% RSLogix 500 project LANLOGIX_BR.RSS, saved by version 12.00.00.00 %
PROJECT "LANLOGIX"    % processor: MicroLogix 1400; MAIN_PROG %

PROGRAM FILES
  LAD 2 "MAIN"  69 rungs
  LAD 4 "MODE SEL"  18 rungs
  LAD 5 "FILM"  6 rungs
  LAD 6 "PROFILES"  56 rungs
  LAD 7 "OPTIONS"  34 rungs
  LAD 8 "CONSTANTS"  5 rungs
  LAD 9 "WRAP CYCLE"  36 rungs
  LAD 10 "OUTPUTS"  46 rungs
  LAD 11 "INPUTS"  77 rungs
  LAD 12 "ROTATION"  44 rungs
  LAD 13 "CARRIAGE"  45 rungs
  LAD 14 "MPS"  23 rungs
  LAD 15 "CUTTER ASM"  18 rungs
  LAD 16 "FILM CLAMP"  15 rungs
  LAD 17 "HOT WIRE"  9 rungs
  LAD 19 "TSD"  37 rungs  % Top Sheet Dispenser %
  LAD 27 "CONV IN 3"  22 rungs
  LAD 28 "CONV IN 2"  22 rungs
  LAD 29 "CONV IN 1"  23 rungs
  LAD 30 "CONV WRAPZ"  29 rungs
  LAD 31 "CONV EX 1"  23 rungs
  LAD 32 "CONV EX 2"  22 rungs
  LAD 33 "CONV EX 3"  22 rungs
  LAD 41 "CONV INTLK"  4 rungs
  LAD 42 "GATE IN"  15 rungs  % Infeed Gate %
  LAD 43 "GATE EX"  15 rungs  % Exit Gate %
  LAD 45 "LOAD LIFT"  12 rungs
  LAD 49 "SECURITY"  11 rungs
  LAD 50 "HMI"  30 rungs
  LAD 52 "CYCLE INFO"  20 rungs
  LAD 98 "WARNINGS"  19 rungs
  LAD 99 "MESSAGES"  28 rungs
  LAD 100 "ALARMS"  36 rungs
  LAD 101 "MAINT"  20 rungs
  LAD 115 "PDATA"  22 rungs  % Production Data %
  LAD 116 "PCHART"  26 rungs  % Production Chart %
  LAD 117 "CDATA"  6 rungs  % Load Containment Data %
  LAD 214 "MPS CALC"  8 rungs
  LAD 250 "VFD MODBUS"  34 rungs
  LAD 251 "MODBUS"  7 rungs
  LAD 255 "HSC PFN"  2 rungs

DATA FILES
  O0 OUTPUT  8 elements
  I1 INPUT  11 elements
  S2 STATUS  66 elements
  B3 BINARY  110 elements
  T4 TIMER  251 elements
  C5 COUNTER  1 elements
  R6 CONTROL  1 elements
  N7 INTEGER  210 elements
  F8 FLOAT  40 elements
  F9 C FORCE  50 elements
  N10 OUTPUT MAP  120 elements
  N11 INPUT MAP  120 elements
  B12 BINARY  120 elements
  B13 BINARY  120 elements
  N14 LG  250 elements
  N15 OPTIONS  15 elements
  N16 SECURITY  10 elements
  N17 MESSAGING  50 elements
  N19 TRACKING  210 elements
  N20 FILM  30 elements
  N21 PROFILES  50 elements
  F22 PROF CALCS  15 elements
  L25 LONG  11 elements
  F26 ICF MAP  16 elements
  N28 TEMP PROF  50 elements  % Temporary Profile %
  N29 INPUT PROF  50 elements  % HMI Input Profile %
  N30 DEFAULT  50 elements  % Default Profile %
  N31 PROFILE 1  50 elements  % Profile 1 %
  N32 PROFILE 2  50 elements  % Profile 2 %
  N33 PROFILE 3  50 elements  % Profile 3 %
  N34 PROFILE 4  50 elements  % Profile 4 %
  N35 PROFILE 5  50 elements  % Profile 5 %
  N36 PROFILE 6  50 elements  % Profile 6 %
  N37 PROFILE 7  50 elements  % Profile 7 %
  N38 PROFILE 8  50 elements  % Profile 8 %
  N39 PROFILE 9  50 elements  % Profile 9 %
  N40 CURRENT  50 elements
  N41 PROFILECAL  28 elements
  ST43 PROFILESTR  10 elements
  ST46 PROFILES  15 elements
  B48 PROF WARN  8 elements
  N49 PROFWARNCH  10 elements
  N50 HMI OUTPUT  256 elements
  N51 HMI INPUT  125 elements
  B60 FAULT  255 elements  % Fault Overflow Trap %
  N80 E_NET_IN  1 elements
  N81 E_NET_OUT  1 elements
  N92 WARNCOPY  10 elements
  N93 WARN BUF  10 elements  % WARNING BUFFER %
  N94 WARN LIST  10 elements  % WARNINGS LIST %
  N95 WARNINGS  10 elements  % WARNINGS %
  N96 ALARMCOPY  50 elements
  N97 ALARM BUF  14 elements  % ALARMS BUFFER %
  N98 ALARM ACT  10 elements  % ALARM ACTIVE %
  N99 ALARM LIST  14 elements  % ALARM LIST %
  N100 ALARMS  50 elements
  N101 MAINT  30 elements
  L102 MAINT1  5 elements
  N103 MAINT2  20 elements
  N110 CDATA  40 elements  % Load Containment Data %
  N111 CDATA1  240 elements  % Load Containment Data Array 1 %
  F112 CDATA2  120 elements  % Load Containment Data Array 2 %
  N115 PDATA  20 elements  % Production Data Control %
  N116 PDATA1  160 elements  % Production Data Array 1 %
  N117 PDATA2  160 elements  % Production Data Array 2 %
  N118 PDATA3  160 elements  % Production Data Array 3 %
  N119 PDATALPH  60 elements  % Production Data Loads/Breaks Per Hour %
  N120 PDATALPR  30 elements  % Production Data Loads Per Film Roll %
  L121 PDATARPR  40 elements  % Production Data Revolutions Per Film Rolls %
  N122 PDATACHART  100 elements  % Production Data Chart %
  N170   3 elements
  N200 MODBUS  50 elements
  MG201 MODBUS MSG  5 elements
  N210 MODBUS OUT  250 elements
  N211 MODBUS IN  250 elements
  ST255 VERSION  1 elements

LADDER 2 "MAIN"
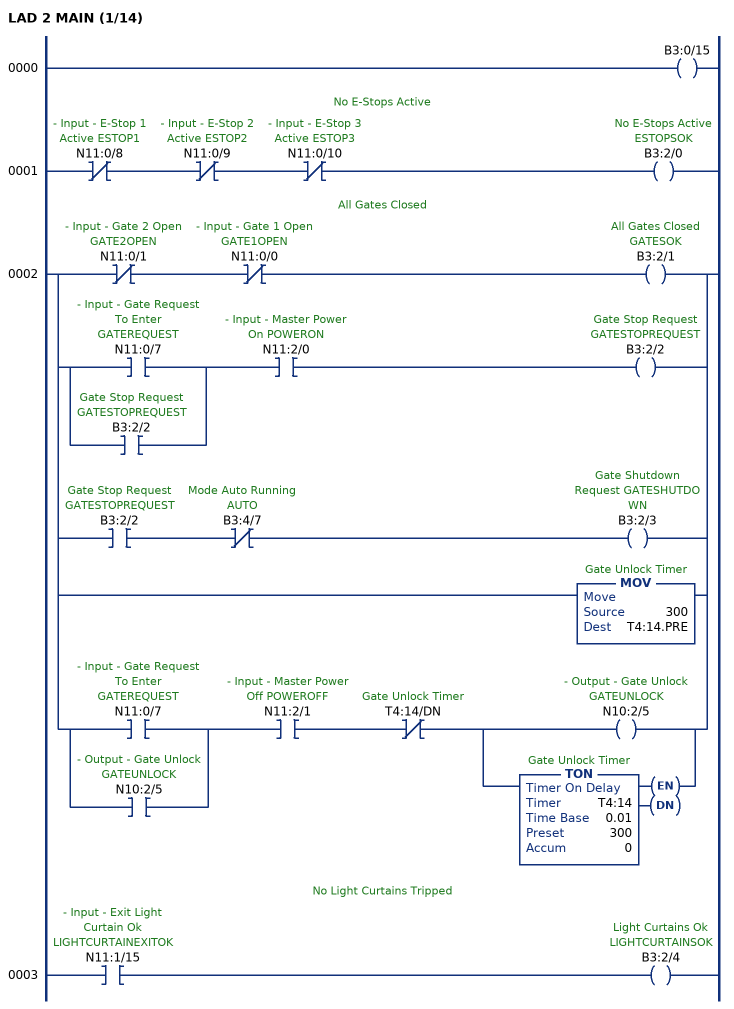
% Rung: 0 %
SOR OTE B3:0/15 EOR
% Rung: 1 %
% No E-Stops Active %
SOR XIO N11:0/8 XIO N11:0/9 XIO N11:0/10 OTE B3:2/0 EOR
%   N11:0/8  ESTOP1  "- Input - E-Stop 1 Active" %
%   N11:0/9  ESTOP2  "- Input - E-Stop 2 Active" %
%   N11:0/10  ESTOP3  "- Input - E-Stop 3 Active" %
%   B3:2/0  ESTOPSOK  "No E-Stops Active" %
% Rung: 2 %
% All Gates Closed %
SOR BST XIO N11:0/1 XIO N11:0/0 OTE B3:2/1 NXB BST XIC N11:0/7 NXB XIC B3:2/2 BND XIC N11:2/0 OTE B3:2/2 NXB XIC B3:2/2 XIO B3:4/7 OTE B3:2/3 NXB MOV 300 T4:14.PRE NXB BST XIC N11:0/7 NXB XIC N10:2/5 BND XIC N11:2/1 XIO T4:14/DN BST OTE N10:2/5 NXB TON T4:14 0.01 300 0 BND BND EOR
%   N11:0/1  GATE2OPEN  "- Input - Gate 2 Open" %
%   N11:0/0  GATE1OPEN  "- Input - Gate 1 Open" %
%   B3:2/1  GATESOK  "All Gates Closed" %
%   N11:0/7  GATEREQUEST  "- Input - Gate Request To Enter" %
%   B3:2/2  GATESTOPREQUEST  "Gate Stop Request" %
%   N11:2/0  POWERON  "- Input - Master Power On" %
%   B3:4/7  AUTO  "Mode Auto Running" %
%   B3:2/3  GATESHUTDOWN  "Gate Shutdown Request" %
%   T4:14  "Gate Unlock Timer" %
%   N10:2/5  GATEUNLOCK  "- Output - Gate Unlock" %
%   N11:2/1  POWEROFF  "- Input - Master Power Off" %
% Rung: 3 %
% No Light Curtains Tripped %
SOR XIC N11:1/15 OTE B3:2/4 EOR
%   N11:1/15  LIGHTCURTAINEXITOK  "- Input - Exit Light Curtain Ok" %
%   B3:2/4  LIGHTCURTAINSOK  "Light Curtains Ok" %

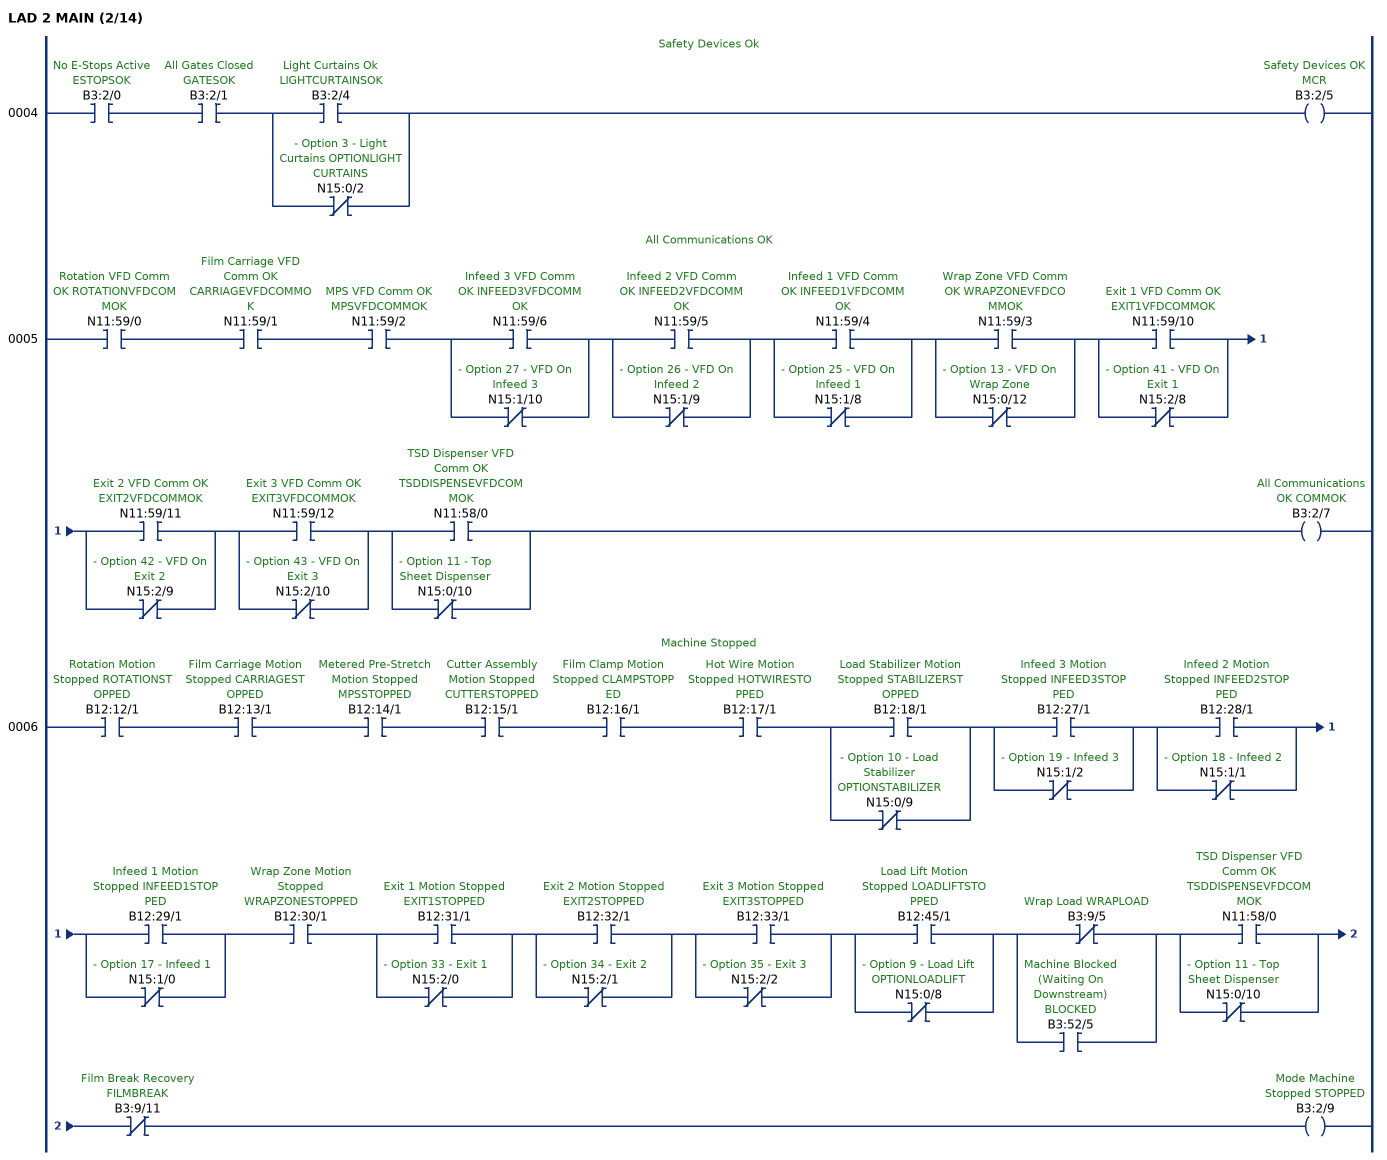
% Rung: 4 %
% Safety Devices Ok %
SOR XIC B3:2/0 XIC B3:2/1 BST XIC B3:2/4 NXB XIO N15:0/2 BND OTE B3:2/5 EOR
%   B3:2/0  ESTOPSOK  "No E-Stops Active" %
%   B3:2/1  GATESOK  "All Gates Closed" %
%   B3:2/4  LIGHTCURTAINSOK  "Light Curtains Ok" %
%   N15:0/2  OPTIONLIGHTCURTAINS  "- Option 3 - Light Curtains" %
%   B3:2/5  MCR  "Safety Devices OK" %
% Rung: 5 %
% All Communications OK %
SOR XIC N11:59/0 XIC N11:59/1 XIC N11:59/2 BST XIC N11:59/6 NXB XIO N15:1/10 BND BST XIC N11:59/5 NXB XIO N15:1/9 BND BST XIC N11:59/4 NXB XIO N15:1/8 BND BST XIC N11:59/3 NXB XIO N15:0/12 BND BST XIC N11:59/10 NXB XIO N15:2/8 BND BST XIC N11:59/11 NXB XIO N15:2/9 BND BST XIC N11:59/12 NXB XIO N15:2/10 BND BST XIC N11:58/0 NXB XIO N15:0/10 BND OTE B3:2/7 EOR
%   N11:59/0  ROTATIONVFDCOMMOK  "Rotation VFD Comm OK" %
%   N11:59/1  CARRIAGEVFDCOMMOK  "Film Carriage VFD Comm OK" %
%   N11:59/2  MPSVFDCOMMOK  "MPS VFD Comm OK" %
%   N11:59/6  INFEED3VFDCOMMOK  "Infeed 3 VFD Comm OK" %
%   N15:1/10  "- Option 27 - VFD On Infeed 3" %
%   N11:59/5  INFEED2VFDCOMMOK  "Infeed 2 VFD Comm OK" %
%   N15:1/9  "- Option 26 - VFD On Infeed 2" %
%   N11:59/4  INFEED1VFDCOMMOK  "Infeed 1 VFD Comm OK" %
%   N15:1/8  "- Option 25 - VFD On Infeed 1" %
%   N11:59/3  WRAPZONEVFDCOMMOK  "Wrap Zone VFD Comm OK" %
%   N15:0/12  "- Option 13 - VFD On Wrap Zone" %
%   N11:59/10  EXIT1VFDCOMMOK  "Exit 1 VFD Comm OK" %
%   N15:2/8  "- Option 41 - VFD On Exit 1" %
%   N11:59/11  EXIT2VFDCOMMOK  "Exit 2 VFD Comm OK" %
%   N15:2/9  "- Option 42 - VFD On Exit 2" %
%   N11:59/12  EXIT3VFDCOMMOK  "Exit 3 VFD Comm OK" %
%   N15:2/10  "- Option 43 - VFD On Exit 3" %
%   N11:58/0  TSDDISPENSEVFDCOMMOK  "TSD Dispenser VFD Comm OK" %
%   N15:0/10  "- Option 11 - Top Sheet Dispenser" %
%   B3:2/7  COMMOK  "All Communications OK" %
% Rung: 6 %
% Machine Stopped %
SOR XIC B12:12/1 XIC B12:13/1 XIC B12:14/1 XIC B12:15/1 XIC B12:16/1 XIC B12:17/1 BST XIC B12:18/1 NXB XIO N15:0/9 BND BST XIC B12:27/1 NXB XIO N15:1/2 BND BST XIC B12:28/1 NXB XIO N15:1/1 BND BST XIC B12:29/1 NXB XIO N15:1/0 BND XIC B12:30/1 BST XIC B12:31/1 NXB XIO N15:2/0 BND BST XIC B12:32/1 NXB XIO N15:2/1 BND BST XIC B12:33/1 NXB XIO N15:2/2 BND BST XIC B12:45/1 NXB XIO N15:0/8 BND BST XIO B3:9/5 NXB XIC B3:52/5 BND BST XIC N11:58/0 NXB XIO N15:0/10 BND XIO B3:9/11 OTE B3:2/9 EOR
%   B12:12/1  ROTATIONSTOPPED  "Rotation Motion Stopped" %
%   B12:13/1  CARRIAGESTOPPED  "Film Carriage Motion Stopped" %
%   B12:14/1  MPSSTOPPED  "Metered Pre-Stretch Motion Stopped" %
%   B12:15/1  CUTTERSTOPPED  "Cutter Assembly Motion Stopped" %
%   B12:16/1  CLAMPSTOPPED  "Film Clamp Motion Stopped" %
%   B12:17/1  HOTWIRESTOPPED  "Hot Wire Motion Stopped" %
%   B12:18/1  STABILIZERSTOPPED  "Load Stabilizer Motion Stopped" %
%   N15:0/9  OPTIONSTABILIZER  "- Option 10 - Load Stabilizer" %
%   B12:27/1  INFEED3STOPPED  "Infeed 3 Motion Stopped" %
%   N15:1/2  "- Option 19 - Infeed 3" %
%   B12:28/1  INFEED2STOPPED  "Infeed 2 Motion Stopped" %
%   N15:1/1  "- Option 18 - Infeed 2" %
%   B12:29/1  INFEED1STOPPED  "Infeed 1 Motion Stopped" %
%   N15:1/0  "- Option 17 - Infeed 1" %
%   B12:30/1  WRAPZONESTOPPED  "Wrap Zone Motion Stopped" %
%   B12:31/1  EXIT1STOPPED  "Exit 1 Motion Stopped" %
%   N15:2/0  "- Option 33 - Exit 1" %
%   B12:32/1  EXIT2STOPPED  "Exit 2 Motion Stopped" %
%   N15:2/1  "- Option 34 - Exit 2" %
%   B12:33/1  EXIT3STOPPED  "Exit 3 Motion Stopped" %
%   N15:2/2  "- Option 35 - Exit 3" %
%   B12:45/1  LOADLIFTSTOPPED  "Load Lift Motion Stopped" %
%   N15:0/8  OPTIONLOADLIFT  "- Option 9 - Load Lift" %
%   B3:9/5  WRAPLOAD  "Wrap Load" %
%   B3:52/5  BLOCKED  "Machine Blocked (Waiting On Downstream)" %
%   N11:58/0  TSDDISPENSEVFDCOMMOK  "TSD Dispenser VFD Comm OK" %
%   N15:0/10  "- Option 11 - Top Sheet Dispenser" %
%   B3:9/11  FILMBREAK  "Film Break Recovery" %
%   B3:2/9  STOPPED  "Mode Machine Stopped" %

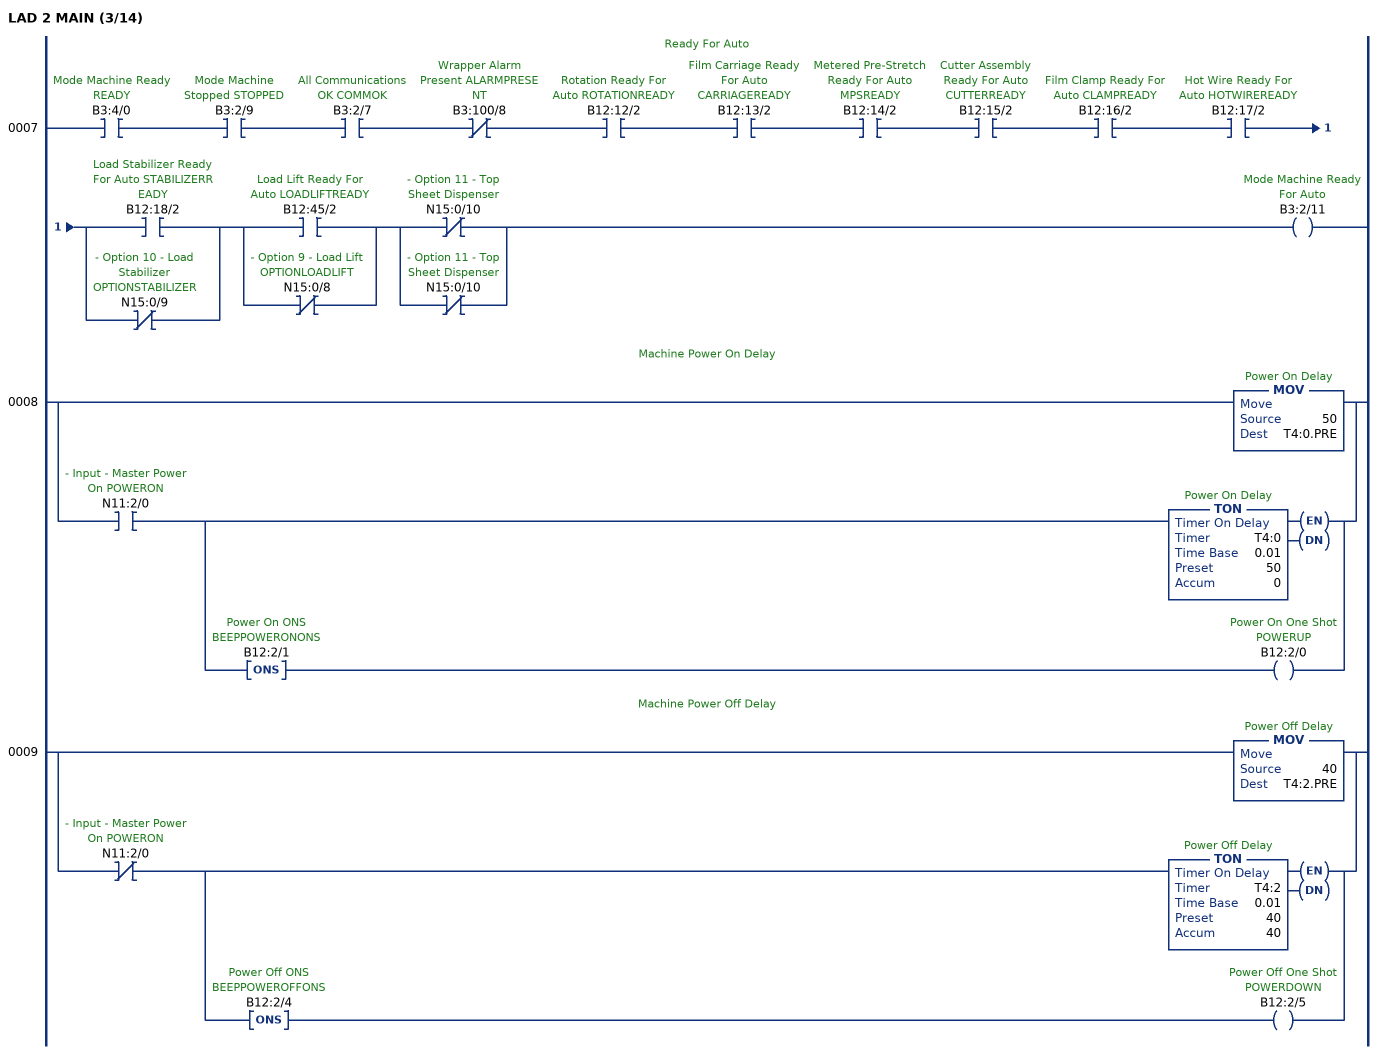
% Rung: 7 %
% Ready For Auto %
SOR XIC B3:4/0 XIC B3:2/9 XIC B3:2/7 XIO B3:100/8 XIC B12:12/2 XIC B12:13/2 XIC B12:14/2 XIC B12:15/2 XIC B12:16/2 XIC B12:17/2 BST XIC B12:18/2 NXB XIO N15:0/9 BND BST XIC B12:45/2 NXB XIO N15:0/8 BND BST XIO N15:0/10 NXB XIO N15:0/10 BND OTE B3:2/11 EOR
%   B3:4/0  READY  "Mode Machine Ready" %
%   B3:2/9  STOPPED  "Mode Machine Stopped" %
%   B3:2/7  COMMOK  "All Communications OK" %
%   B3:100/8  ALARMPRESENT  "Wrapper Alarm Present" %
%   B12:12/2  ROTATIONREADY  "Rotation Ready For Auto" %
%   B12:13/2  CARRIAGEREADY  "Film Carriage Ready For Auto" %
%   B12:14/2  MPSREADY  "Metered Pre-Stretch Ready For Auto" %
%   B12:15/2  CUTTERREADY  "Cutter Assembly Ready For Auto" %
%   B12:16/2  CLAMPREADY  "Film Clamp Ready For Auto" %
%   B12:17/2  HOTWIREREADY  "Hot Wire Ready For Auto" %
%   B12:18/2  STABILIZERREADY  "Load Stabilizer Ready For Auto" %
%   N15:0/9  OPTIONSTABILIZER  "- Option 10 - Load Stabilizer" %
%   B12:45/2  LOADLIFTREADY  "Load Lift Ready For Auto" %
%   N15:0/8  OPTIONLOADLIFT  "- Option 9 - Load Lift" %
%   N15:0/10  "- Option 11 - Top Sheet Dispenser" %
%   B3:2/11  "Mode Machine Ready For Auto" %
% Rung: 8 %
% Machine Power On Delay %
SOR BST MOV 50 T4:0.PRE NXB XIC N11:2/0 BST TON T4:0 0.01 50 0 NXB ONS B12:2/1 OTE B12:2/0 BND BND EOR
%   T4:0  "Power On Delay" %
%   N11:2/0  POWERON  "- Input - Master Power On" %
%   B12:2/1  BEEPPOWERONONS  "Power On ONS" %
%   B12:2/0  POWERUP  "Power On One Shot" %
% Rung: 9 %
% Machine Power Off Delay %
SOR BST MOV 40 T4:2.PRE NXB XIO N11:2/0 BST TON T4:2 0.01 40 40 NXB ONS B12:2/4 OTE B12:2/5 BND BND EOR
%   T4:2  "Power Off Delay" %
%   N11:2/0  POWERON  "- Input - Master Power On" %
%   B12:2/4  BEEPPOWEROFFONS  "Power Off ONS" %
%   B12:2/5  POWERDOWN  "Power Off One Shot" %

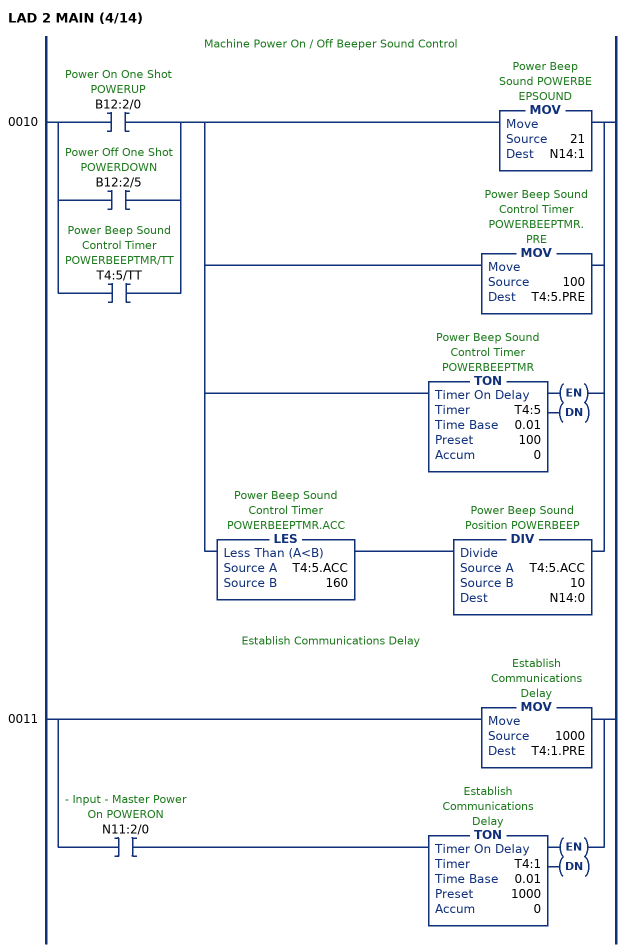
% Rung: 10 %
% Machine Power On / Off Beeper Sound Control %
SOR BST XIC B12:2/0 NXB XIC B12:2/5 NXB XIC T4:5/TT BND BST MOV 21 N14:1 NXB MOV 100 T4:5.PRE NXB TON T4:5 0.01 100 0 NXB LES T4:5.ACC 160 DIV T4:5.ACC 10 N14:0 BND EOR
%   B12:2/0  POWERUP  "Power On One Shot" %
%   B12:2/5  POWERDOWN  "Power Off One Shot" %
%   T4:5  POWERBEEPTMR  "Power Beep Sound Control Timer" %
%   N14:1  POWERBEEPSOUND  "Power Beep Sound" %
%   N14:0  POWERBEEP  "Power Beep Sound Position" %
% Rung: 11 %
% Establish Communications Delay %
SOR BST MOV 1000 T4:1.PRE NXB XIC N11:2/0 TON T4:1 0.01 1000 0 BND EOR
%   T4:1  "Establish Communications Delay" %
%   N11:2/0  POWERON  "- Input - Master Power On" %

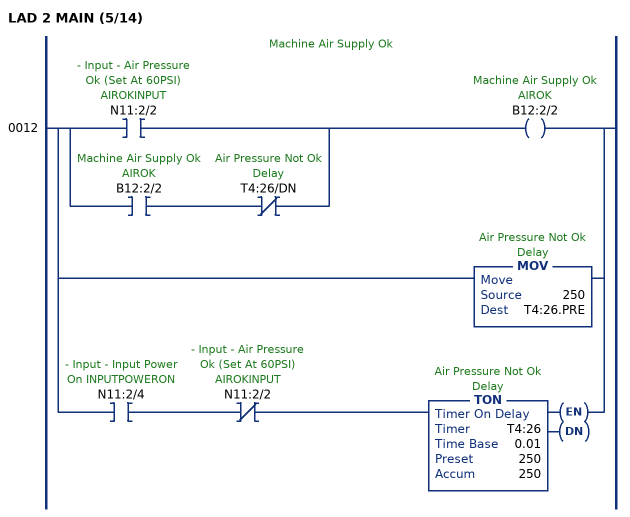
% Rung: 12 %
% Machine Air Supply Ok %
SOR BST BST XIC N11:2/2 NXB XIC B12:2/2 XIO T4:26/DN BND OTE B12:2/2 NXB MOV 250 T4:26.PRE NXB XIC N11:2/4 XIO N11:2/2 TON T4:26 0.01 250 250 BND EOR
%   N11:2/2  AIROKINPUT  "- Input - Air Pressure Ok (Set At 60PSI)" %
%   B12:2/2  AIROK  "Machine Air Supply Ok" %
%   T4:26  "Air Pressure Not Ok Delay" %
%   N11:2/4  INPUTPOWERON  "- Input - Input Power On" %

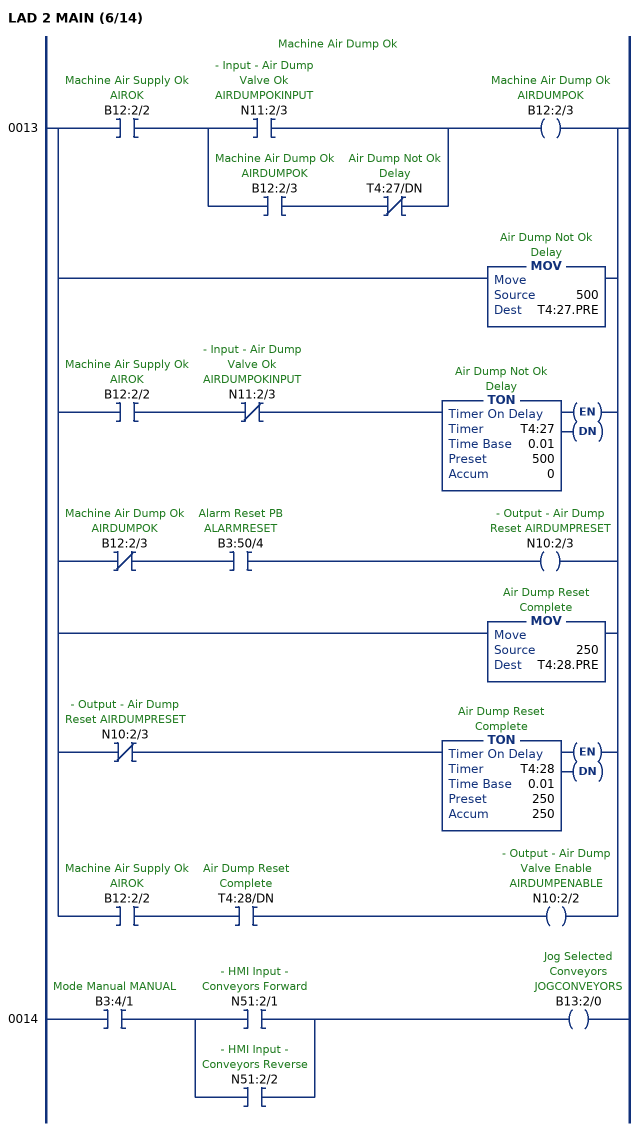
% Rung: 13 %
% Machine Air Dump Ok %
SOR BST XIC B12:2/2 BST XIC N11:2/3 NXB XIC B12:2/3 XIO T4:27/DN BND OTE B12:2/3 NXB MOV 500 T4:27.PRE NXB XIC B12:2/2 XIO N11:2/3 TON T4:27 0.01 500 0 NXB XIO B12:2/3 XIC B3:50/4 OTE N10:2/3 NXB MOV 250 T4:28.PRE NXB XIO N10:2/3 TON T4:28 0.01 250 250 NXB XIC B12:2/2 XIC T4:28/DN OTE N10:2/2 BND EOR
%   B12:2/2  AIROK  "Machine Air Supply Ok" %
%   N11:2/3  AIRDUMPOKINPUT  "- Input - Air Dump Valve Ok" %
%   B12:2/3  AIRDUMPOK  "Machine Air Dump Ok" %
%   T4:27  "Air Dump Not Ok Delay" %
%   B3:50/4  ALARMRESET  "Alarm Reset PB" %
%   N10:2/3  AIRDUMPRESET  "- Output - Air Dump Reset" %
%   T4:28  "Air Dump Reset Complete" %
%   N10:2/2  AIRDUMPENABLE  "- Output - Air Dump Valve Enable" %
% Rung: 14 %
SOR XIC B3:4/1 BST XIC N51:2/1 NXB XIC N51:2/2 BND OTE B13:2/0 EOR
%   B3:4/1  MANUAL  "Mode Manual" %
%   N51:2/1  "- HMI Input - Conveyors Forward" %
%   N51:2/2  "- HMI Input - Conveyors Reverse" %
%   B13:2/0  JOGCONVEYORS  "Jog Selected Conveyors" %

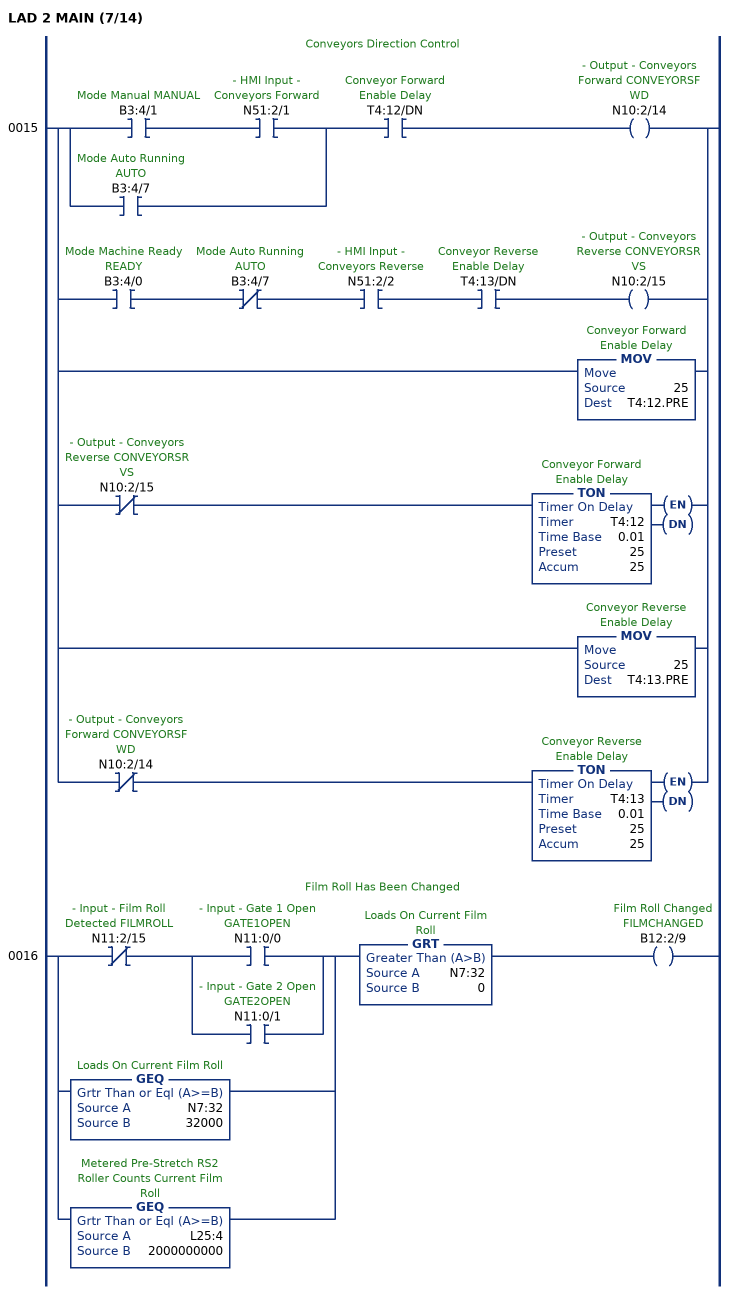
% Rung: 15 %
% Conveyors Direction Control %
SOR BST BST XIC B3:4/1 XIC N51:2/1 NXB XIC B3:4/7 BND XIC T4:12/DN OTE N10:2/14 NXB XIC B3:4/0 XIO B3:4/7 XIC N51:2/2 XIC T4:13/DN OTE N10:2/15 NXB MOV 25 T4:12.PRE NXB XIO N10:2/15 TON T4:12 0.01 25 25 NXB MOV 25 T4:13.PRE NXB XIO N10:2/14 TON T4:13 0.01 25 25 BND EOR
%   B3:4/1  MANUAL  "Mode Manual" %
%   N51:2/1  "- HMI Input - Conveyors Forward" %
%   B3:4/7  AUTO  "Mode Auto Running" %
%   T4:12  "Conveyor Forward Enable Delay" %
%   N10:2/14  CONVEYORSFWD  "- Output - Conveyors Forward" %
%   B3:4/0  READY  "Mode Machine Ready" %
%   N51:2/2  "- HMI Input - Conveyors Reverse" %
%   T4:13  "Conveyor Reverse Enable Delay" %
%   N10:2/15  CONVEYORSRVS  "- Output - Conveyors Reverse" %
% Rung: 16 %
% Film Roll Has Been Changed %
SOR BST XIO N11:2/15 BST XIC N11:0/0 NXB XIC N11:0/1 BND NXB GEQ N7:32 32000 NXB GEQ L25:4 2000000000 BND GRT N7:32 0 OTE B12:2/9 EOR
%   N11:2/15  FILMROLL  "- Input - Film Roll Detected" %
%   N11:0/0  GATE1OPEN  "- Input - Gate 1 Open" %
%   N11:0/1  GATE2OPEN  "- Input - Gate 2 Open" %
%   N7:32  "Loads On Current Film Roll" %
%   L25:4  "Metered Pre-Stretch RS2 Roller Counts Current Film Roll" %
%   B12:2/9  FILMCHANGED  "Film Roll Changed" %

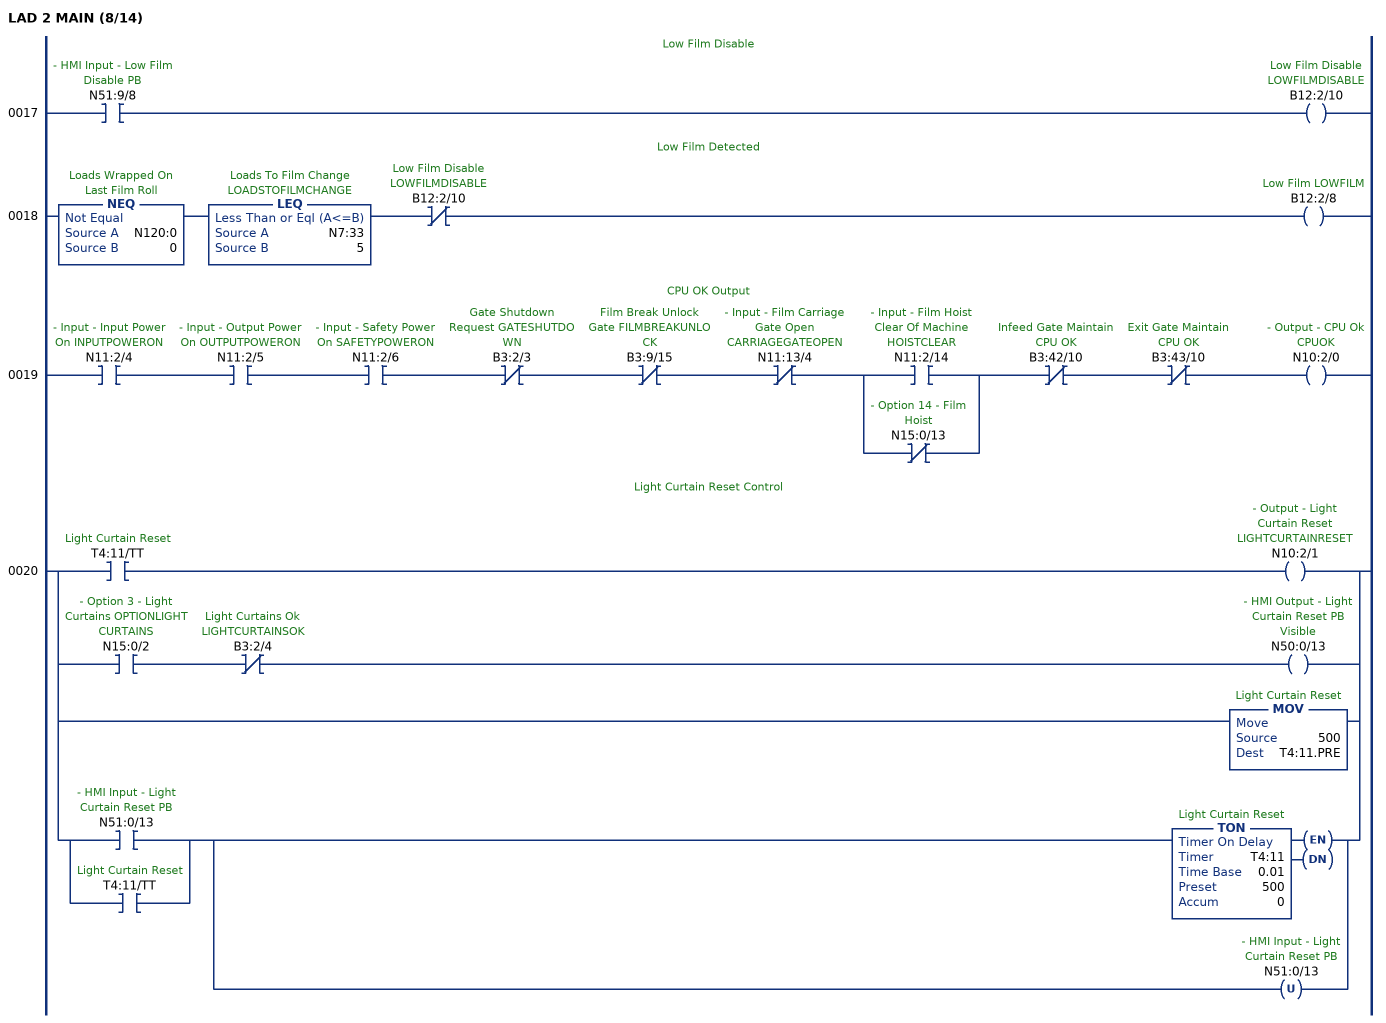
% Rung: 17 %
% Low Film Disable %
SOR XIC N51:9/8 OTE B12:2/10 EOR
%   N51:9/8  "- HMI Input - Low Film Disable PB" %
%   B12:2/10  LOWFILMDISABLE  "Low Film Disable" %
% Rung: 18 %
% Low Film Detected %
SOR NEQ N120:0 0 LEQ N7:33 5 XIO B12:2/10 OTE B12:2/8 EOR
%   N120:0  "Loads Wrapped On Last Film Roll" %
%   N7:33  LOADSTOFILMCHANGE  "Loads To Film Change" %
%   B12:2/10  LOWFILMDISABLE  "Low Film Disable" %
%   B12:2/8  LOWFILM  "Low Film" %
% Rung: 19 %
% CPU OK Output %
SOR XIC N11:2/4 XIC N11:2/5 XIC N11:2/6 XIO B3:2/3 XIO B3:9/15 XIO N11:13/4 BST XIC N11:2/14 NXB XIO N15:0/13 BND XIO B3:42/10 XIO B3:43/10 OTE N10:2/0 EOR
%   N11:2/4  INPUTPOWERON  "- Input - Input Power On" %
%   N11:2/5  OUTPUTPOWERON  "- Input - Output Power On" %
%   N11:2/6  SAFETYPOWERON  "- Input - Safety Power On" %
%   B3:2/3  GATESHUTDOWN  "Gate Shutdown Request" %
%   B3:9/15  FILMBREAKUNLOCK  "Film Break Unlock Gate" %
%   N11:13/4  CARRIAGEGATEOPEN  "- Input - Film Carriage Gate Open" %
%   N11:2/14  HOISTCLEAR  "- Input - Film Hoist Clear Of Machine" %
%   N15:0/13  "- Option 14 - Film Hoist" %
%   B3:42/10  "Infeed Gate Maintain CPU OK" %
%   B3:43/10  "Exit Gate Maintain CPU OK" %
%   N10:2/0  CPUOK  "- Output - CPU Ok" %
% Rung: 20 %
% Light Curtain Reset Control %
SOR BST XIC T4:11/TT OTE N10:2/1 NXB XIC N15:0/2 XIO B3:2/4 OTE N50:0/13 NXB MOV 500 T4:11.PRE NXB BST XIC N51:0/13 NXB XIC T4:11/TT BND BST TON T4:11 0.01 500 0 NXB OTU N51:0/13 BND BND EOR
%   T4:11  "Light Curtain Reset" %
%   N10:2/1  LIGHTCURTAINRESET  "- Output - Light Curtain Reset" %
%   N15:0/2  OPTIONLIGHTCURTAINS  "- Option 3 - Light Curtains" %
%   B3:2/4  LIGHTCURTAINSOK  "Light Curtains Ok" %
%   N50:0/13  "- HMI Output - Light Curtain Reset PB Visible" %
%   N51:0/13  "- HMI Input - Light Curtain Reset PB" %

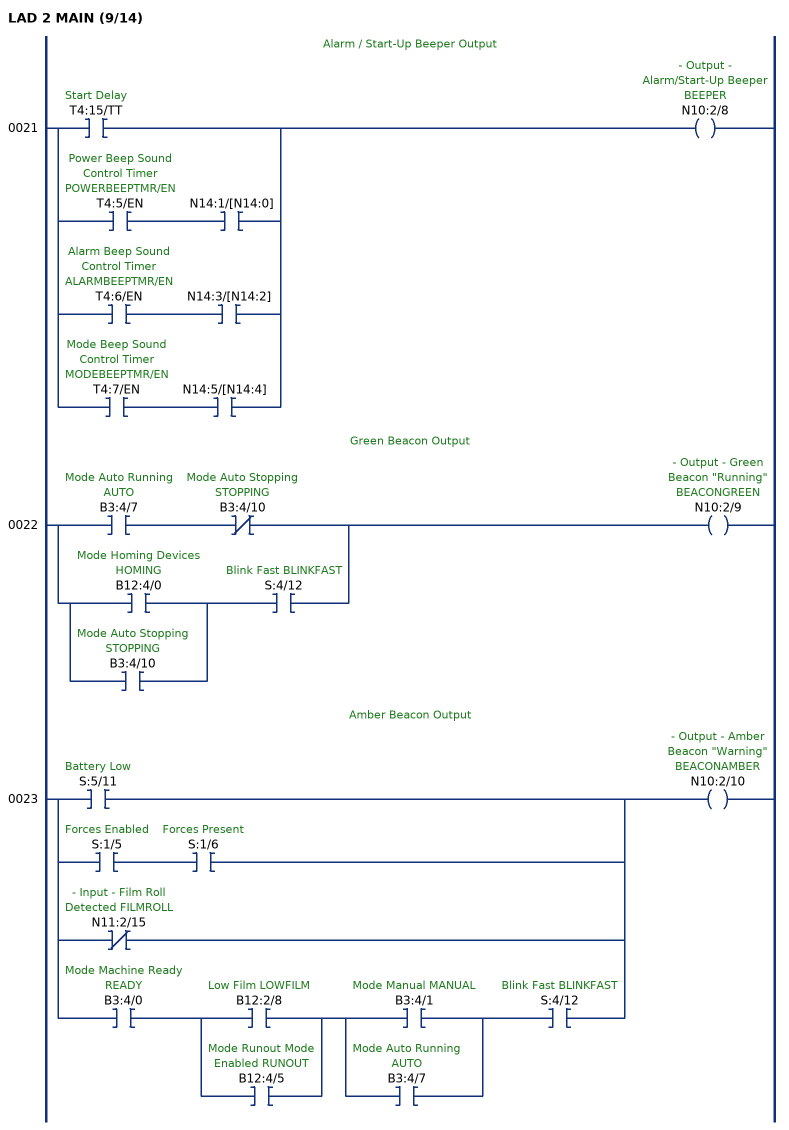
% Rung: 21 %
% Alarm / Start-Up Beeper Output %
SOR BST XIC T4:15/TT NXB XIC T4:5/EN XIC N14:1/[N14:0] NXB XIC T4:6/EN XIC N14:3/[N14:2] NXB XIC T4:7/EN XIC N14:5/[N14:4] BND OTE N10:2/8 EOR
%   T4:15  "Start Delay" %
%   T4:5  POWERBEEPTMR  "Power Beep Sound Control Timer" %
%   N14:1  POWERBEEPSOUND  "Power Beep Sound" %
%   N14:0  POWERBEEP  "Power Beep Sound Position" %
%   T4:6  ALARMBEEPTMR  "Alarm Beep Sound Control Timer" %
%   N14:3  ALARMBEEPSOUND  "Alarm Beep Sound" %
%   N14:2  ALARMBEEP  "Alarm Beep Soud Position" %
%   T4:7  MODEBEEPTMR  "Mode Beep Sound Control Timer" %
%   N14:5  MODEBEEPSOUND  "Mode Beep Sound" %
%   N14:4  MODEBEEP  "Mode Beep Sound Position" %
%   N10:2/8  BEEPER  "- Output - Alarm/Start-Up Beeper" %
% Rung: 22 %
% Green Beacon Output %
SOR BST XIC B3:4/7 XIO B3:4/10 NXB BST XIC B12:4/0 NXB XIC B3:4/10 BND XIC S:4/12 BND OTE N10:2/9 EOR
%   B3:4/7  AUTO  "Mode Auto Running" %
%   B3:4/10  STOPPING  "Mode Auto Stopping" %
%   B12:4/0  HOMING  "Mode Homing Devices" %
%   S:4/12  BLINKFAST  "Blink Fast" %
%   N10:2/9  BEACONGREEN  "- Output - Green Beacon "Running"" %
% Rung: 23 %
% Amber Beacon Output %
SOR BST XIC S:5/11 NXB XIC S:1/5 XIC S:1/6 NXB XIO N11:2/15 NXB XIC B3:4/0 BST XIC B12:2/8 NXB XIC B12:4/5 BND BST XIC B3:4/1 NXB XIC B3:4/7 BND XIC S:4/12 BND OTE N10:2/10 EOR
%   S:5/11  "Battery Low" %
%   S:1/5  "Forces Enabled" %
%   S:1/6  "Forces Present" %
%   N11:2/15  FILMROLL  "- Input - Film Roll Detected" %
%   B3:4/0  READY  "Mode Machine Ready" %
%   B12:2/8  LOWFILM  "Low Film" %
%   B12:4/5  RUNOUT  "Mode Runout Mode Enabled" %
%   B3:4/1  MANUAL  "Mode Manual" %
%   B3:4/7  AUTO  "Mode Auto Running" %
%   S:4/12  BLINKFAST  "Blink Fast" %
%   N10:2/10  BEACONAMBER  "- Output - Amber Beacon "Warning"" %

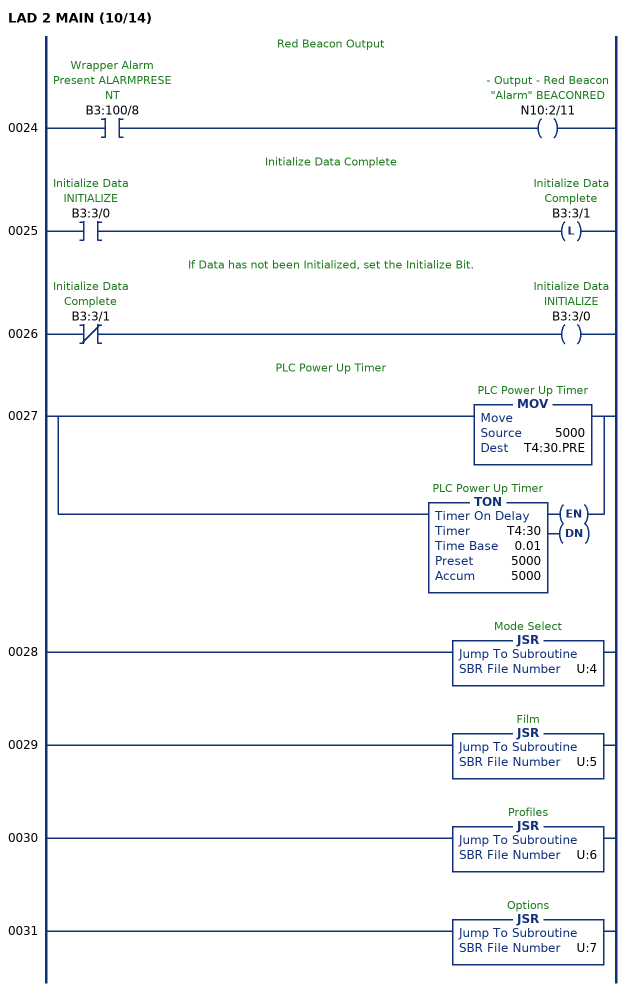
% Rung: 24 %
% Red Beacon Output %
SOR XIC B3:100/8 OTE N10:2/11 EOR
%   B3:100/8  ALARMPRESENT  "Wrapper Alarm Present" %
%   N10:2/11  BEACONRED  "- Output - Red Beacon "Alarm"" %
% Rung: 25 %
% Initialize Data Complete %
SOR XIC B3:3/0 OTL B3:3/1 EOR
%   B3:3/0  INITIALIZE  "Initialize Data" %
%   B3:3/1  "Initialize Data Complete" %
% Rung: 26 %
% If Data has not been Initialized, set the Initialize Bit. %
SOR XIO B3:3/1 OTE B3:3/0 EOR
%   B3:3/1  "Initialize Data Complete" %
%   B3:3/0  INITIALIZE  "Initialize Data" %
% Rung: 27 %
% PLC Power Up Timer %
SOR BST MOV 5000 T4:30.PRE NXB TON T4:30 0.01 5000 5000 BND EOR
%   T4:30  "PLC Power Up Timer" %
% Rung: 28 %
SOR JSR U:4 EOR
%   U:4  "Mode Select" %
% Rung: 29 %
SOR JSR U:5 EOR
%   U:5  "Film" %
% Rung: 30 %
SOR JSR U:6 EOR
%   U:6  "Profiles" %
% Rung: 31 %
SOR JSR U:7 EOR
%   U:7  "Options" %

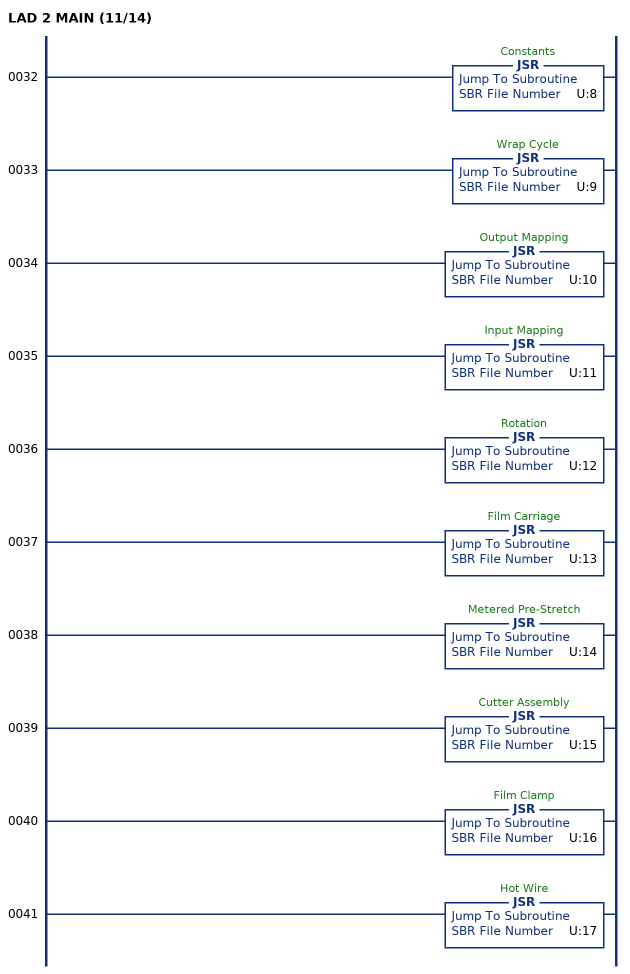
% Rung: 32 %
SOR JSR U:8 EOR
%   U:8  "Constants" %
% Rung: 33 %
SOR JSR U:9 EOR
%   U:9  "Wrap Cycle" %
% Rung: 34 %
SOR JSR U:10 EOR
%   U:10  "Output Mapping" %
% Rung: 35 %
SOR JSR U:11 EOR
%   U:11  "Input Mapping" %
% Rung: 36 %
SOR JSR U:12 EOR
%   U:12  "Rotation" %
% Rung: 37 %
SOR JSR U:13 EOR
%   U:13  "Film Carriage" %
% Rung: 38 %
SOR JSR U:14 EOR
%   U:14  "Metered Pre-Stretch" %
% Rung: 39 %
SOR JSR U:15 EOR
%   U:15  "Cutter Assembly" %
% Rung: 40 %
SOR JSR U:16 EOR
%   U:16  "Film Clamp" %
% Rung: 41 %
SOR JSR U:17 EOR
%   U:17  "Hot Wire" %

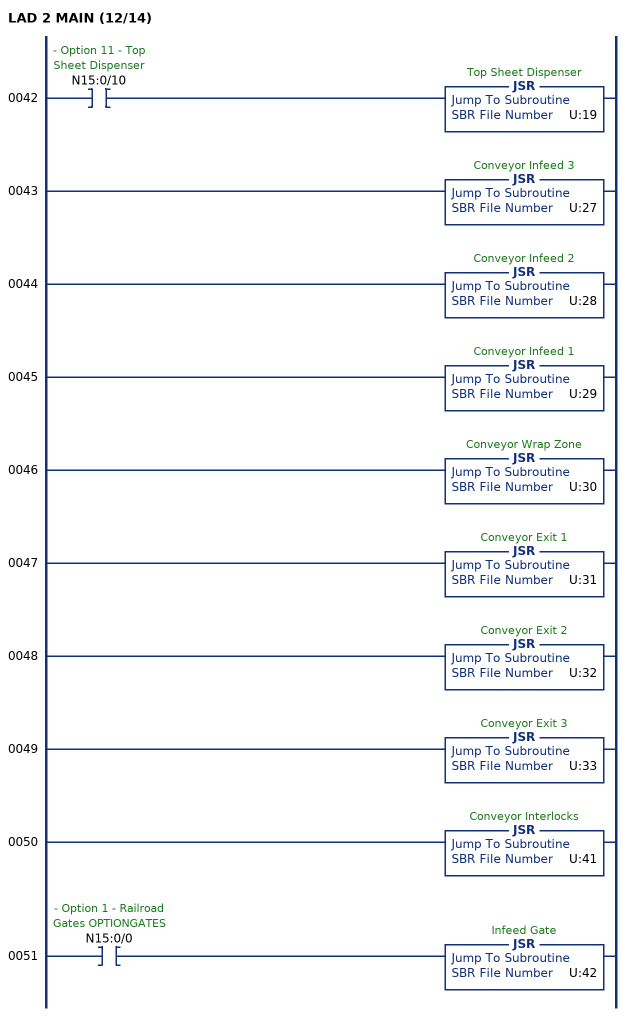
% Rung: 42 %
SOR XIC N15:0/10 JSR U:19 EOR
%   N15:0/10  "- Option 11 - Top Sheet Dispenser" %
%   U:19  "Top Sheet Dispenser" %
% Rung: 43 %
SOR JSR U:27 EOR
%   U:27  "Conveyor Infeed 3" %
% Rung: 44 %
SOR JSR U:28 EOR
%   U:28  "Conveyor Infeed 2" %
% Rung: 45 %
SOR JSR U:29 EOR
%   U:29  "Conveyor Infeed 1" %
% Rung: 46 %
SOR JSR U:30 EOR
%   U:30  "Conveyor Wrap Zone" %
% Rung: 47 %
SOR JSR U:31 EOR
%   U:31  "Conveyor Exit 1" %
% Rung: 48 %
SOR JSR U:32 EOR
%   U:32  "Conveyor Exit 2" %
% Rung: 49 %
SOR JSR U:33 EOR
%   U:33  "Conveyor Exit 3" %
% Rung: 50 %
SOR JSR U:41 EOR
%   U:41  "Conveyor Interlocks" %
% Rung: 51 %
SOR XIC N15:0/0 JSR U:42 EOR
%   N15:0/0  OPTIONGATES  "- Option 1 - Railroad Gates" %
%   U:42  "Infeed Gate" %

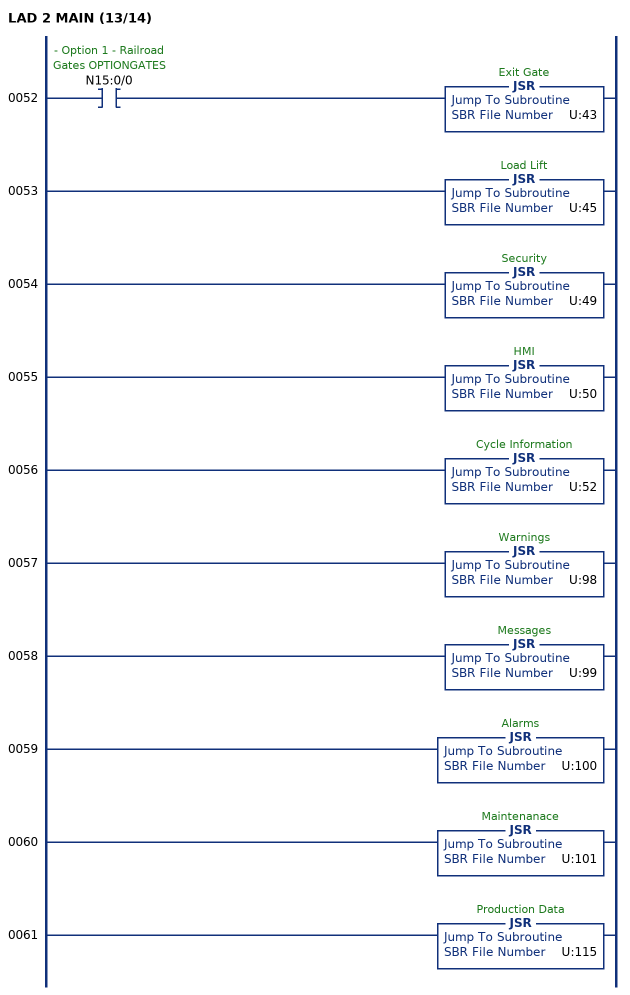
% Rung: 52 %
SOR XIC N15:0/0 JSR U:43 EOR
%   N15:0/0  OPTIONGATES  "- Option 1 - Railroad Gates" %
%   U:43  "Exit Gate" %
% Rung: 53 %
SOR JSR U:45 EOR
%   U:45  "Load Lift" %
% Rung: 54 %
SOR JSR U:49 EOR
%   U:49  "Security" %
% Rung: 55 %
SOR JSR U:50 EOR
%   U:50  "HMI" %
% Rung: 56 %
SOR JSR U:52 EOR
%   U:52  "Cycle Information" %
% Rung: 57 %
SOR JSR U:98 EOR
%   U:98  "Warnings" %
% Rung: 58 %
SOR JSR U:99 EOR
%   U:99  "Messages" %
% Rung: 59 %
SOR JSR U:100 EOR
%   U:100  "Alarms" %
% Rung: 60 %
SOR JSR U:101 EOR
%   U:101  "Maintenanace" %
% Rung: 61 %
SOR JSR U:115 EOR
%   U:115  "Production Data" %

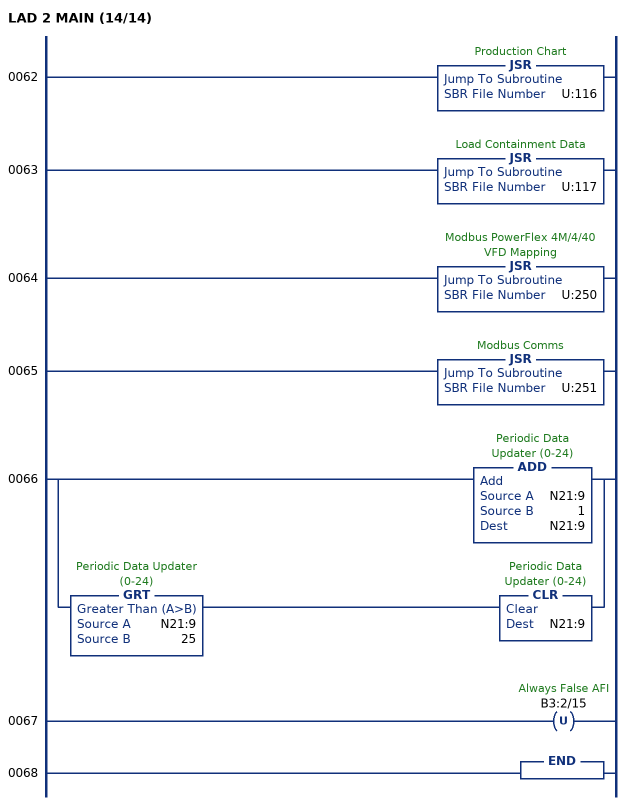
% Rung: 62 %
SOR JSR U:116 EOR
%   U:116  "Production Chart" %
% Rung: 63 %
SOR JSR U:117 EOR
%   U:117  "Load Containment Data" %
% Rung: 64 %
SOR JSR U:250 EOR
%   U:250  "Modbus PowerFlex 4M/4/40 VFD Mapping" %
% Rung: 65 %
SOR JSR U:251 EOR
%   U:251  "Modbus Comms" %
% Rung: 66 %
SOR BST ADD N21:9 1 N21:9 NXB GRT N21:9 25 CLR N21:9 BND EOR
%   N21:9  "Periodic Data Updater (0-24)" %
% Rung: 67 %
SOR OTU B3:2/15 EOR
%   B3:2/15  AFI  "Always False" %
% Rung: 68 %
SOR END EOR

LADDER 4 "MODE SEL"
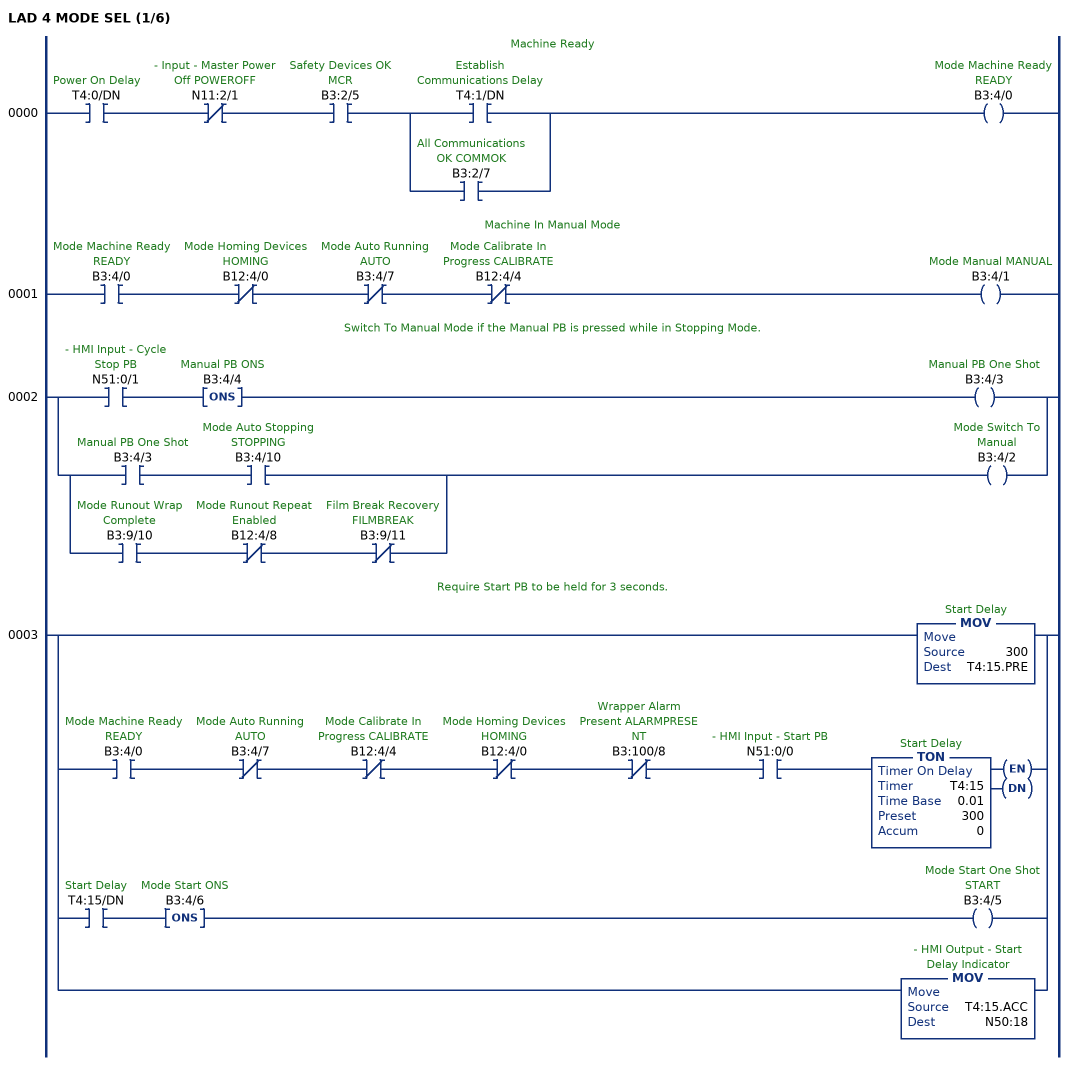
% Rung: 0 %
% Machine Ready %
SOR XIC T4:0/DN XIO N11:2/1 XIC B3:2/5 BST XIC T4:1/DN NXB XIC B3:2/7 BND OTE B3:4/0 EOR
%   T4:0  "Power On Delay" %
%   N11:2/1  POWEROFF  "- Input - Master Power Off" %
%   B3:2/5  MCR  "Safety Devices OK" %
%   T4:1  "Establish Communications Delay" %
%   B3:2/7  COMMOK  "All Communications OK" %
%   B3:4/0  READY  "Mode Machine Ready" %
% Rung: 1 %
% Machine In Manual Mode %
SOR XIC B3:4/0 XIO B12:4/0 XIO B3:4/7 XIO B12:4/4 OTE B3:4/1 EOR
%   B3:4/0  READY  "Mode Machine Ready" %
%   B12:4/0  HOMING  "Mode Homing Devices" %
%   B3:4/7  AUTO  "Mode Auto Running" %
%   B12:4/4  CALIBRATE  "Mode Calibrate In Progress" %
%   B3:4/1  MANUAL  "Mode Manual" %
% Rung: 2 %
% Switch To Manual Mode if the Manual PB is pressed while in Stopping Mode. %
SOR BST XIC N51:0/1 ONS B3:4/4 OTE B3:4/3 NXB BST XIC B3:4/3 XIC B3:4/10 NXB XIC B3:9/10 XIO B12:4/8 XIO B3:9/11 BND OTE B3:4/2 BND EOR
%   N51:0/1  "- HMI Input - Cycle Stop PB" %
%   B3:4/4  "Manual PB ONS" %
%   B3:4/3  "Manual PB One Shot" %
%   B3:4/10  STOPPING  "Mode Auto Stopping" %
%   B3:9/10  "Mode Runout Wrap Complete" %
%   B12:4/8  "Mode Runout Repeat Enabled" %
%   B3:9/11  FILMBREAK  "Film Break Recovery" %
%   B3:4/2  "Mode Switch To Manual" %
% Rung: 3 %
% Require Start PB to be held for 3 seconds. %
SOR BST MOV 300 T4:15.PRE NXB XIC B3:4/0 XIO B3:4/7 XIO B12:4/4 XIO B12:4/0 XIO B3:100/8 XIC N51:0/0 TON T4:15 0.01 300 0 NXB XIC T4:15/DN ONS B3:4/6 OTE B3:4/5 NXB MOV T4:15.ACC N50:18 BND EOR
%   T4:15  "Start Delay" %
%   B3:4/0  READY  "Mode Machine Ready" %
%   B3:4/7  AUTO  "Mode Auto Running" %
%   B12:4/4  CALIBRATE  "Mode Calibrate In Progress" %
%   B12:4/0  HOMING  "Mode Homing Devices" %
%   B3:100/8  ALARMPRESENT  "Wrapper Alarm Present" %
%   N51:0/0  "- HMI Input - Start PB" %
%   B3:4/6  "Mode Start ONS" %
%   B3:4/5  START  "Mode Start One Shot" %
%   N50:18  "- HMI Output - Start Delay Indicator" %

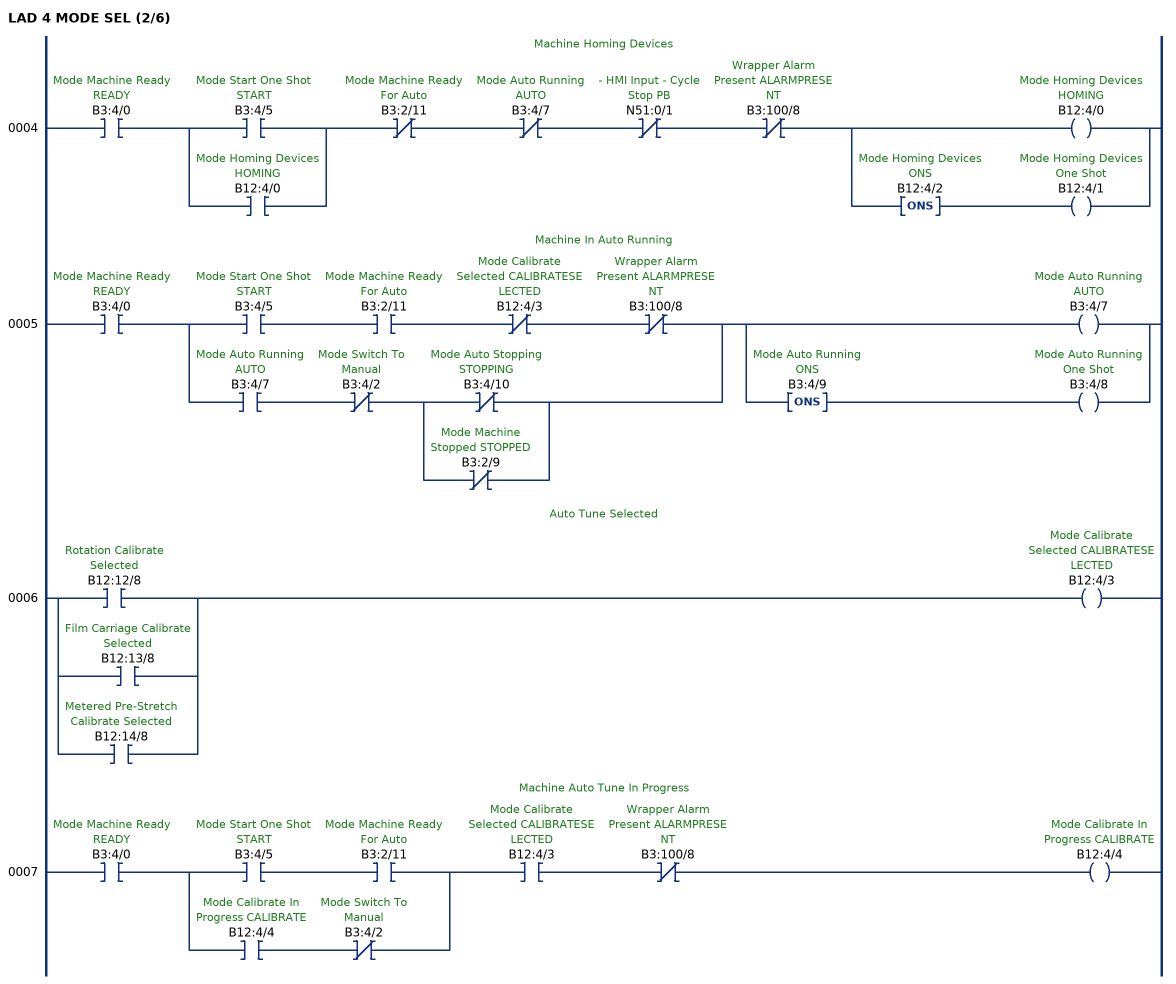
% Rung: 4 %
% Machine Homing Devices %
SOR XIC B3:4/0 BST XIC B3:4/5 NXB XIC B12:4/0 BND XIO B3:2/11 XIO B3:4/7 XIO N51:0/1 XIO B3:100/8 BST OTE B12:4/0 NXB ONS B12:4/2 OTE B12:4/1 BND EOR
%   B3:4/0  READY  "Mode Machine Ready" %
%   B3:4/5  START  "Mode Start One Shot" %
%   B12:4/0  HOMING  "Mode Homing Devices" %
%   B3:2/11  "Mode Machine Ready For Auto" %
%   B3:4/7  AUTO  "Mode Auto Running" %
%   N51:0/1  "- HMI Input - Cycle Stop PB" %
%   B3:100/8  ALARMPRESENT  "Wrapper Alarm Present" %
%   B12:4/2  "Mode Homing Devices ONS" %
%   B12:4/1  "Mode Homing Devices One Shot" %
% Rung: 5 %
% Machine In Auto Running %
SOR XIC B3:4/0 BST XIC B3:4/5 XIC B3:2/11 XIO B12:4/3 XIO B3:100/8 NXB XIC B3:4/7 XIO B3:4/2 BST XIO B3:4/10 NXB XIO B3:2/9 BND BND BST OTE B3:4/7 NXB ONS B3:4/9 OTE B3:4/8 BND EOR
%   B3:4/0  READY  "Mode Machine Ready" %
%   B3:4/5  START  "Mode Start One Shot" %
%   B3:2/11  "Mode Machine Ready For Auto" %
%   B12:4/3  CALIBRATESELECTED  "Mode Calibrate Selected" %
%   B3:100/8  ALARMPRESENT  "Wrapper Alarm Present" %
%   B3:4/7  AUTO  "Mode Auto Running" %
%   B3:4/2  "Mode Switch To Manual" %
%   B3:4/10  STOPPING  "Mode Auto Stopping" %
%   B3:2/9  STOPPED  "Mode Machine Stopped" %
%   B3:4/9  "Mode Auto Running ONS" %
%   B3:4/8  "Mode Auto Running One Shot" %
% Rung: 6 %
% Auto Tune Selected %
SOR BST XIC B12:12/8 NXB XIC B12:13/8 NXB XIC B12:14/8 BND OTE B12:4/3 EOR
%   B12:12/8  "Rotation Calibrate Selected" %
%   B12:13/8  "Film Carriage Calibrate Selected" %
%   B12:14/8  "Metered Pre-Stretch Calibrate Selected" %
%   B12:4/3  CALIBRATESELECTED  "Mode Calibrate Selected" %
% Rung: 7 %
% Machine Auto Tune In Progress %
SOR XIC B3:4/0 BST XIC B3:4/5 XIC B3:2/11 NXB XIC B12:4/4 XIO B3:4/2 BND XIC B12:4/3 XIO B3:100/8 OTE B12:4/4 EOR
%   B3:4/0  READY  "Mode Machine Ready" %
%   B3:4/5  START  "Mode Start One Shot" %
%   B3:2/11  "Mode Machine Ready For Auto" %
%   B12:4/4  CALIBRATE  "Mode Calibrate In Progress" %
%   B3:4/2  "Mode Switch To Manual" %
%   B12:4/3  CALIBRATESELECTED  "Mode Calibrate Selected" %
%   B3:100/8  ALARMPRESENT  "Wrapper Alarm Present" %

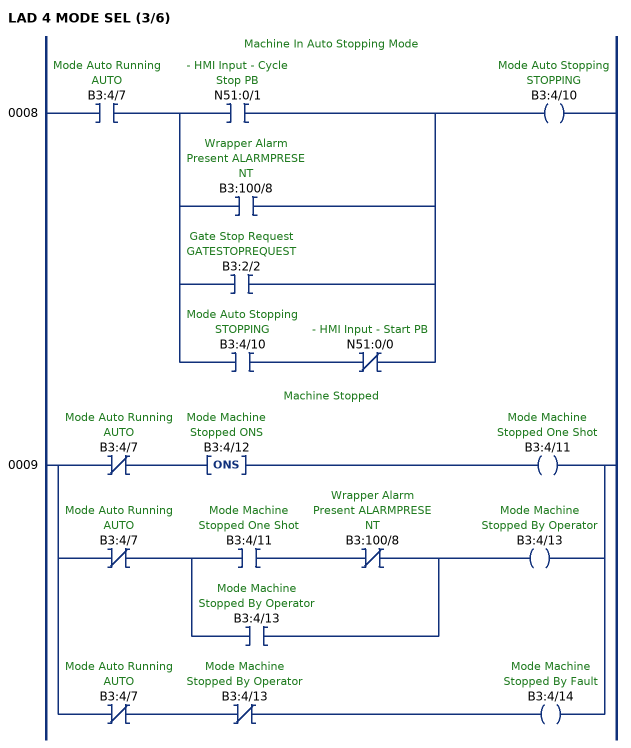
% Rung: 8 %
% Machine In Auto Stopping Mode %
SOR XIC B3:4/7 BST XIC N51:0/1 NXB XIC B3:100/8 NXB XIC B3:2/2 NXB XIC B3:4/10 XIO N51:0/0 BND OTE B3:4/10 EOR
%   B3:4/7  AUTO  "Mode Auto Running" %
%   N51:0/1  "- HMI Input - Cycle Stop PB" %
%   B3:100/8  ALARMPRESENT  "Wrapper Alarm Present" %
%   B3:2/2  GATESTOPREQUEST  "Gate Stop Request" %
%   B3:4/10  STOPPING  "Mode Auto Stopping" %
%   N51:0/0  "- HMI Input - Start PB" %
% Rung: 9 %
% Machine Stopped %
SOR BST XIO B3:4/7 ONS B3:4/12 OTE B3:4/11 NXB XIO B3:4/7 BST XIC B3:4/11 XIO B3:100/8 NXB XIC B3:4/13 BND OTE B3:4/13 NXB XIO B3:4/7 XIO B3:4/13 OTE B3:4/14 BND EOR
%   B3:4/7  AUTO  "Mode Auto Running" %
%   B3:4/12  "Mode Machine Stopped ONS" %
%   B3:4/11  "Mode Machine Stopped One Shot" %
%   B3:100/8  ALARMPRESENT  "Wrapper Alarm Present" %
%   B3:4/13  "Mode Machine Stopped By Operator" %
%   B3:4/14  "Mode Machine Stopped By Fault" %

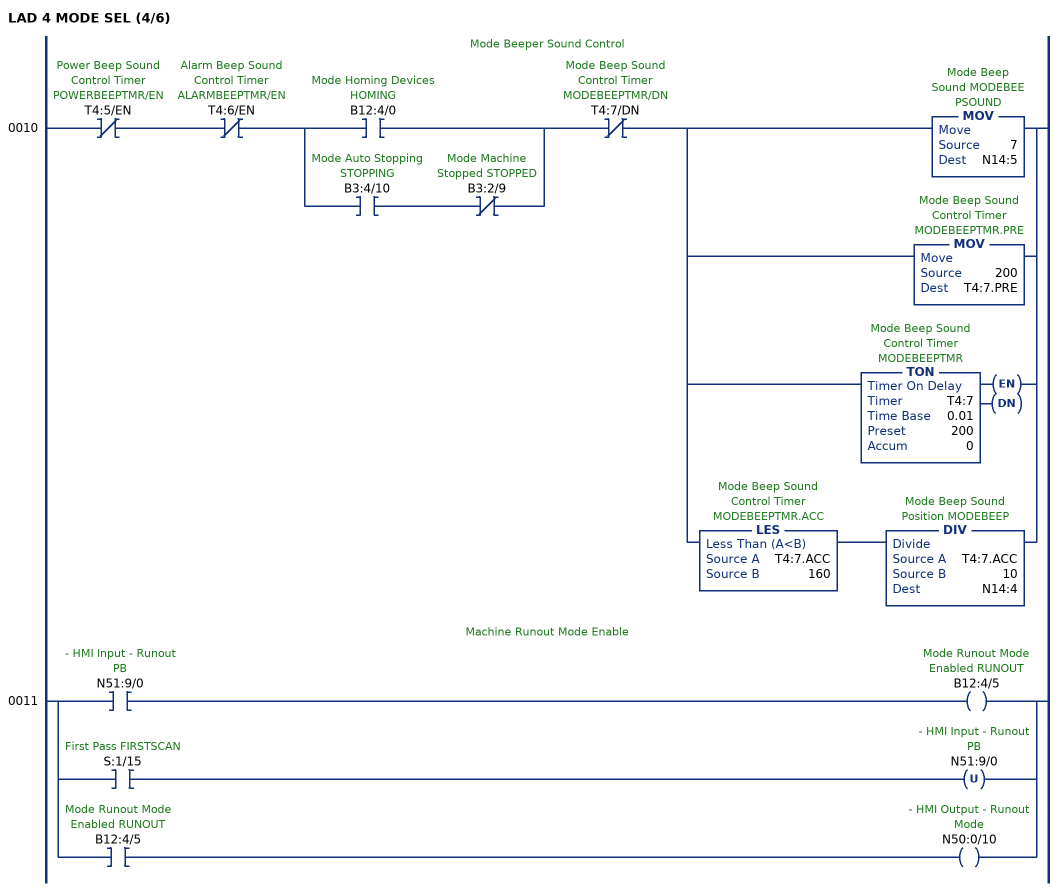
% Rung: 10 %
% Mode Beeper Sound Control %
SOR XIO T4:5/EN XIO T4:6/EN BST XIC B12:4/0 NXB XIC B3:4/10 XIO B3:2/9 BND XIO T4:7/DN BST MOV 7 N14:5 NXB MOV 200 T4:7.PRE NXB TON T4:7 0.01 200 0 NXB LES T4:7.ACC 160 DIV T4:7.ACC 10 N14:4 BND EOR
%   T4:5  POWERBEEPTMR  "Power Beep Sound Control Timer" %
%   T4:6  ALARMBEEPTMR  "Alarm Beep Sound Control Timer" %
%   B12:4/0  HOMING  "Mode Homing Devices" %
%   B3:4/10  STOPPING  "Mode Auto Stopping" %
%   B3:2/9  STOPPED  "Mode Machine Stopped" %
%   T4:7  MODEBEEPTMR  "Mode Beep Sound Control Timer" %
%   N14:5  MODEBEEPSOUND  "Mode Beep Sound" %
%   N14:4  MODEBEEP  "Mode Beep Sound Position" %
% Rung: 11 %
% Machine Runout Mode Enable %
SOR BST XIC N51:9/0 OTE B12:4/5 NXB XIC S:1/15 OTU N51:9/0 NXB XIC B12:4/5 OTE N50:0/10 BND EOR
%   N51:9/0  "- HMI Input - Runout PB" %
%   B12:4/5  RUNOUT  "Mode Runout Mode Enabled" %
%   S:1/15  FIRSTSCAN  "First Pass" %
%   N50:0/10  "- HMI Output - Runout Mode" %

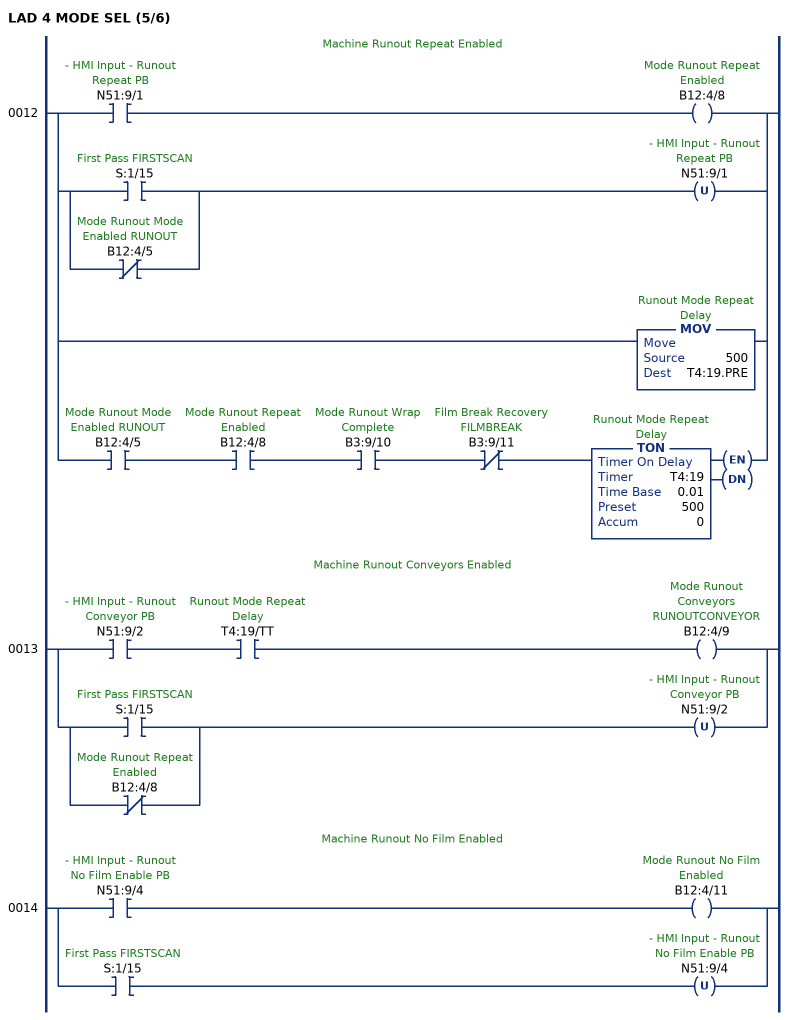
% Rung: 12 %
% Machine Runout Repeat Enabled %
SOR BST XIC N51:9/1 OTE B12:4/8 NXB BST XIC S:1/15 NXB XIO B12:4/5 BND OTU N51:9/1 NXB MOV 500 T4:19.PRE NXB XIC B12:4/5 XIC B12:4/8 XIC B3:9/10 XIO B3:9/11 TON T4:19 0.01 500 0 BND EOR
%   N51:9/1  "- HMI Input - Runout Repeat PB" %
%   B12:4/8  "Mode Runout Repeat Enabled" %
%   S:1/15  FIRSTSCAN  "First Pass" %
%   B12:4/5  RUNOUT  "Mode Runout Mode Enabled" %
%   T4:19  "Runout Mode Repeat Delay" %
%   B3:9/10  "Mode Runout Wrap Complete" %
%   B3:9/11  FILMBREAK  "Film Break Recovery" %
% Rung: 13 %
% Machine Runout Conveyors Enabled %
SOR BST XIC N51:9/2 XIC T4:19/TT OTE B12:4/9 NXB BST XIC S:1/15 NXB XIO B12:4/8 BND OTU N51:9/2 BND EOR
%   N51:9/2  "- HMI Input - Runout Conveyor PB" %
%   T4:19  "Runout Mode Repeat Delay" %
%   B12:4/9  RUNOUTCONVEYOR  "Mode Runout Conveyors" %
%   S:1/15  FIRSTSCAN  "First Pass" %
%   B12:4/8  "Mode Runout Repeat Enabled" %
% Rung: 14 %
% Machine Runout No Film Enabled %
SOR BST XIC N51:9/4 OTE B12:4/11 NXB XIC S:1/15 OTU N51:9/4 BND EOR
%   N51:9/4  "- HMI Input - Runout No Film Enable PB" %
%   B12:4/11  "Mode Runout No Film Enabled" %
%   S:1/15  FIRSTSCAN  "First Pass" %

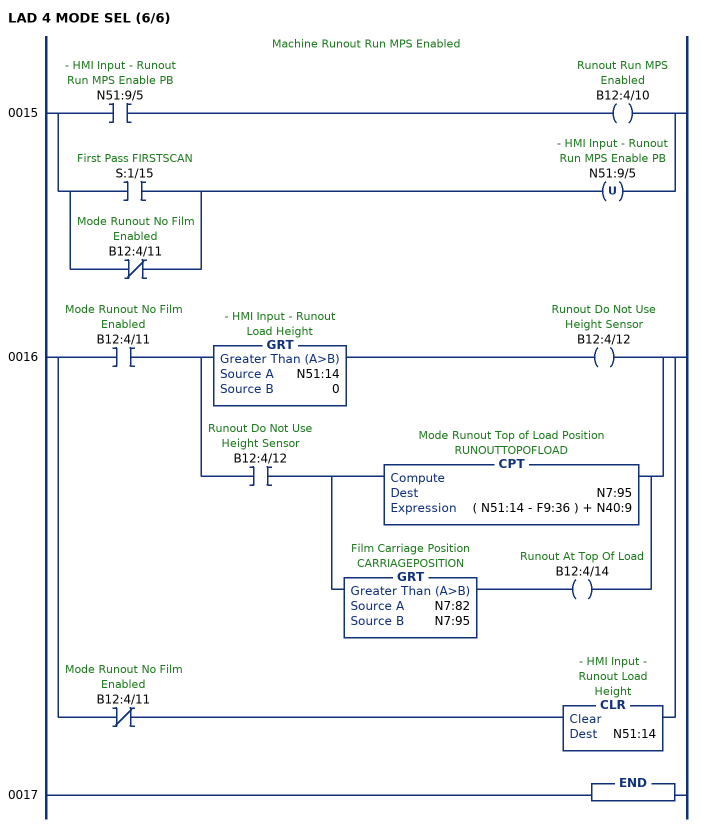
% Rung: 15 %
% Machine Runout Run MPS Enabled %
SOR BST XIC N51:9/5 OTE B12:4/10 NXB BST XIC S:1/15 NXB XIO B12:4/11 BND OTU N51:9/5 BND EOR
%   N51:9/5  "- HMI Input - Runout Run MPS Enable PB" %
%   B12:4/10  "Runout Run MPS Enabled" %
%   S:1/15  FIRSTSCAN  "First Pass" %
%   B12:4/11  "Mode Runout No Film Enabled" %
% Rung: 16 %
SOR BST XIC B12:4/11 BST GRT N51:14 0 OTE B12:4/12 NXB XIC B12:4/12 BST CPT N7:95 " ( N51:14 - F9:36 ) + N40:9 " NXB GRT N7:82 N7:95 OTE B12:4/14 BND BND NXB XIO B12:4/11 CLR N51:14 BND EOR
%   B12:4/11  "Mode Runout No Film Enabled" %
%   N51:14  "- HMI Input - Runout Load Height" %
%   B12:4/12  "Runout Do Not Use Height Sensor" %
%   N7:95  RUNOUTTOPOFLOAD  "Mode Runout Top of Load Position" %
%   F9:36  FILMWIDTHATLOAD  "Film Width At Load" %
%   N40:9  "Current Profile Top Overwrap (Inches)" %
%   N7:82  CARRIAGEPOSITION  "Film Carriage Position" %
%   B12:4/14  "Runout At Top Of Load" %
% Rung: 17 %
SOR END EOR

LADDER 5 "FILM"
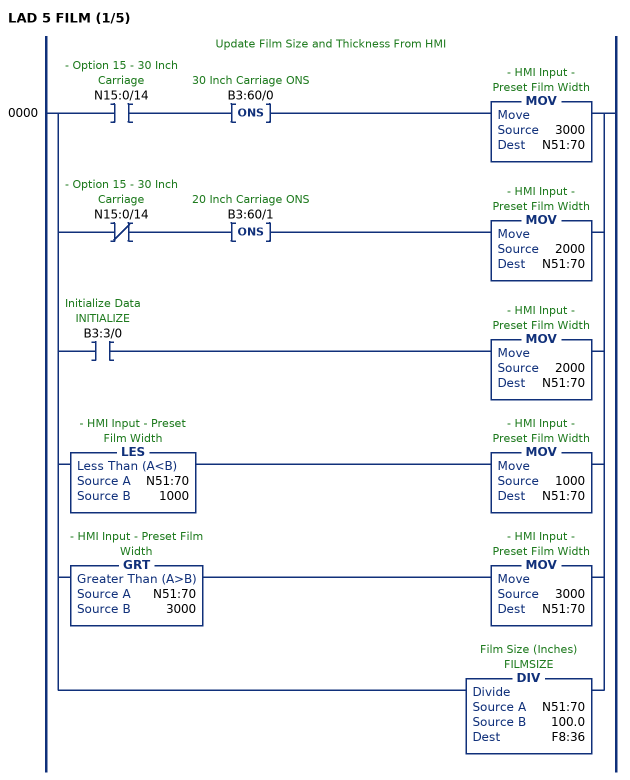
% Rung: 0 %
% Update Film Size and Thickness From HMI %
SOR BST XIC N15:0/14 ONS B3:60/0 MOV 3000 N51:70 NXB XIO N15:0/14 ONS B3:60/1 MOV 2000 N51:70 NXB BST XIC B3:3/0 MOV 2000 N51:70 NXB LES N51:70 1000 MOV 1000 N51:70 NXB GRT N51:70 3000 MOV 3000 N51:70 NXB DIV N51:70 100.0 F8:36 BND BND EOR
%   N15:0/14  "- Option 15 - 30 Inch Carriage" %
%   B3:60/0  "30 Inch Carriage ONS" %
%   N51:70  "- HMI Input - Preset Film Width" %
%   B3:60/1  "20 Inch Carriage ONS" %
%   B3:3/0  INITIALIZE  "Initialize Data" %
%   F8:36  FILMSIZE  "Film Size (Inches)" %

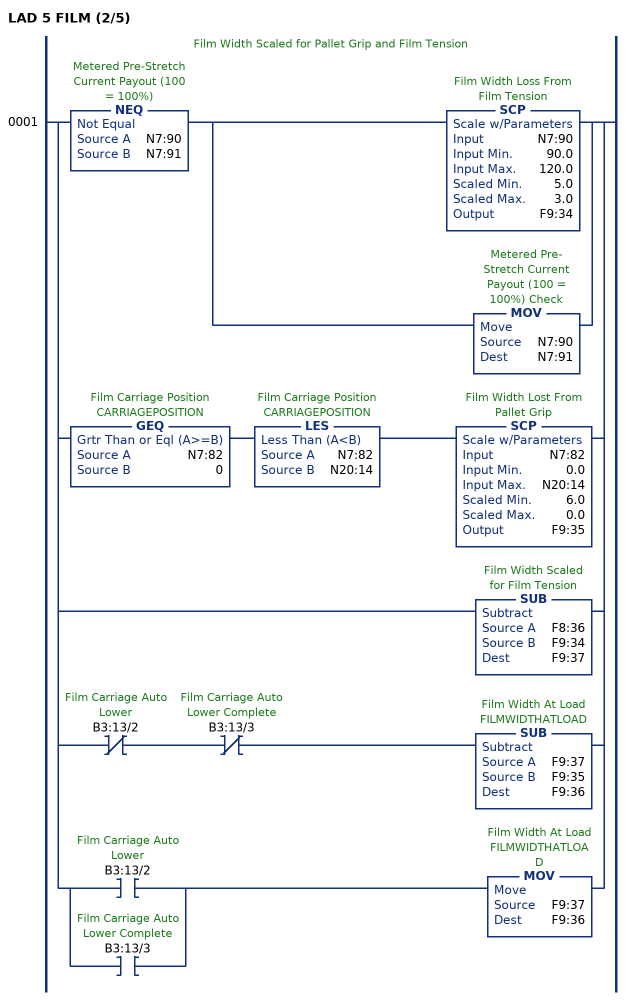
% Rung: 1 %
% Film Width Scaled for Pallet Grip and Film Tension %
SOR BST NEQ N7:90 N7:91 BST SCP N7:90 90.0 120.0 5.0 3.0 F9:34 NXB MOV N7:90 N7:91 BND NXB GEQ N7:82 0 LES N7:82 N20:14 SCP N7:82 0.0 N20:14 6.0 0.0 F9:35 NXB SUB F8:36 F9:34 F9:37 NXB XIO B3:13/2 XIO B3:13/3 SUB F9:37 F9:35 F9:36 NXB BST XIC B3:13/2 NXB XIC B3:13/3 BND MOV F9:37 F9:36 BND EOR
%   N7:90  "Metered Pre-Stretch Current Payout (100 = 100%)" %
%   N7:91  "Metered Pre-Stretch Current Payout (100 = 100%) Check" %
%   F9:34  "Film Width Loss From Film Tension" %
%   N7:82  CARRIAGEPOSITION  "Film Carriage Position" %
%   N20:14  "Pallet-Grip Fully Released Position (10 = 10 Inches)" %
%   F9:35  "Film Width Lost From Pallet Grip" %
%   F8:36  FILMSIZE  "Film Size (Inches)" %
%   F9:37  "Film Width Scaled for Film Tension" %
%   B3:13/2  "Film Carriage Auto Lower" %
%   B3:13/3  "Film Carriage Auto Lower Complete" %
%   F9:36  FILMWIDTHATLOAD  "Film Width At Load" %

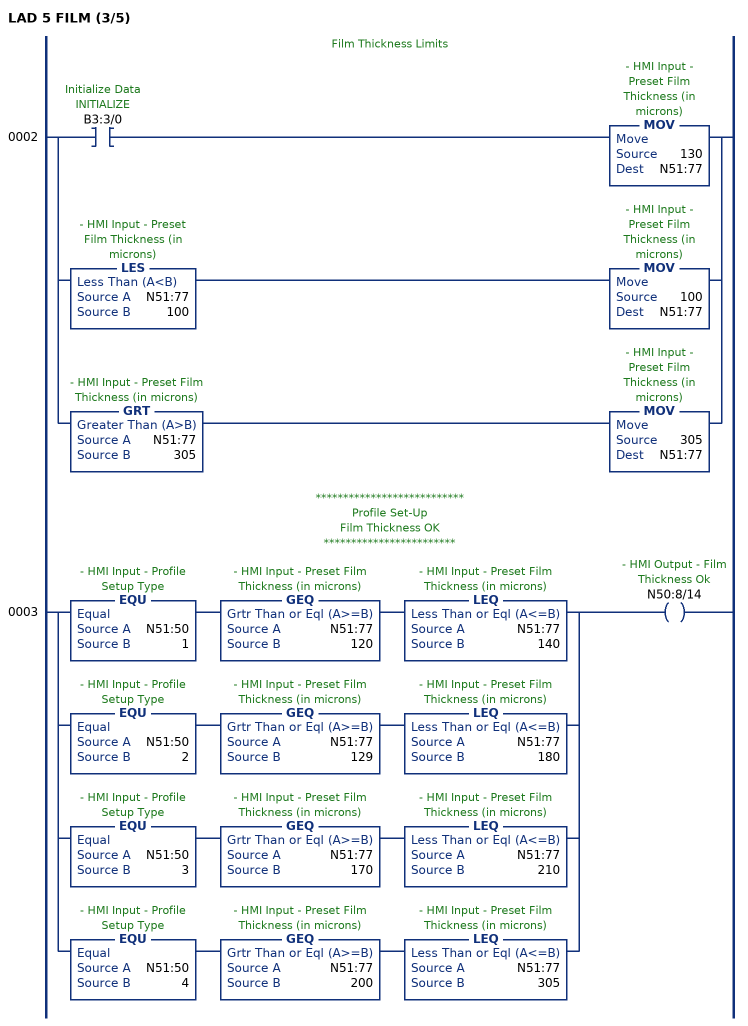
% Rung: 2 %
% Film Thickness Limits %
SOR BST XIC B3:3/0 MOV 130 N51:77 NXB LES N51:77 100 MOV 100 N51:77 NXB GRT N51:77 305 MOV 305 N51:77 BND EOR
%   B3:3/0  INITIALIZE  "Initialize Data" %
%   N51:77  "- HMI Input - Preset Film Thickness (in microns)" %
% Rung: 3 %
% ***************************
% 
% Profile Set-Up
% Film Thickness OK
% 
% ************************ %
SOR BST EQU N51:50 1 GEQ N51:77 120 LEQ N51:77 140 NXB EQU N51:50 2 GEQ N51:77 129 LEQ N51:77 180 NXB EQU N51:50 3 GEQ N51:77 170 LEQ N51:77 210 NXB EQU N51:50 4 GEQ N51:77 200 LEQ N51:77 305 BND OTE N50:8/14 EOR
%   N51:50  "- HMI Input - Profile Setup Type" %
%   N51:77  "- HMI Input - Preset Film Thickness (in microns)" %
%   N50:8/14  "- HMI Output - Film Thickness Ok" %

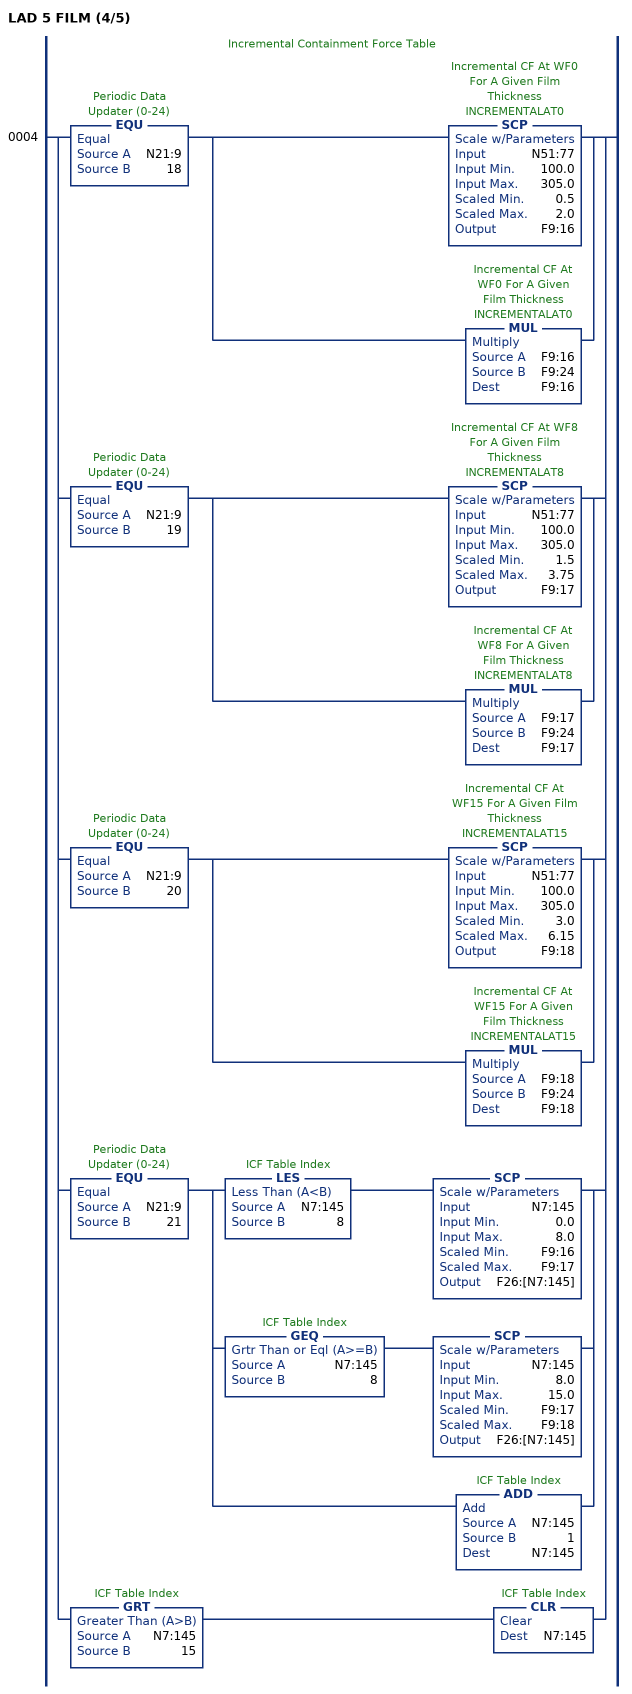
% Rung: 4 %
% Incremental Containment Force Table %
SOR BST BST EQU N21:9 18 BST SCP N51:77 100.0 305.0 0.5 2.0 F9:16 NXB MUL F9:16 F9:24 F9:16 BND NXB EQU N21:9 19 BST SCP N51:77 100.0 305.0 1.5 3.75 F9:17 NXB MUL F9:17 F9:24 F9:17 BND NXB EQU N21:9 20 BST SCP N51:77 100.0 305.0 3.0 6.15 F9:18 NXB MUL F9:18 F9:24 F9:18 BND BND NXB EQU N21:9 21 BST LES N7:145 8 SCP N7:145 0.0 8.0 F9:16 F9:17 F26:[N7:145] NXB GEQ N7:145 8 SCP N7:145 8.0 15.0 F9:17 F9:18 F26:[N7:145] NXB ADD N7:145 1 N7:145 BND NXB GRT N7:145 15 CLR N7:145 BND EOR
%   N21:9  "Periodic Data Updater (0-24)" %
%   N51:77  "- HMI Input - Preset Film Thickness (in microns)" %
%   F9:16  INCREMENTALAT0  "Incremental CF At WF0 For A Given Film Thickness" %
%   F9:24  CALIBRATIONMUL  "Calibration Multiplier" %
%   F9:17  INCREMENTALAT8  "Incremental CF At WF8 For A Given Film Thickness" %
%   F9:18  INCREMENTALAT15  "Incremental CF At WF15 For A Given Film Thickness" %
%   N7:145  "ICF Table Index" %

